LIN {X 0,Y 357.465,Z 383.249,A -85,B 0,C 180,E1 -13742.726,E2 -13742.726} C_VEL
LIN {X 0,Y 362.153,Z 407.547,A -85,B 0,C 180,E1 -13743.635,E2 -13743.635} C_VEL
LIN {X 0,Y 359.928,Z 505.63,A -85,B 0,C 180,E1 -13745.602,E2 -13745.602} C_VEL
LIN {X 0,Y 359.113,Z 520.358,A -85,B 0,C 180,E1 -13746.081,E2 -13746.081} C_VEL
LIN {X 0,Y 358.08,Z 533.693,A -85,B 0,C 180,E1 -13746.737,E2 -13746.737} C_VEL
LIN {X 0,Y 356.818,Z 546.527,A -85,B 0,C 180,E1 -13747.584,E2 -13747.584} C_VEL
LIN {X 0,Y 355.315,Z 560.099,A -85,B 0,C 180,E1 -13748.756,E2 -13748.756} C_VEL
LIN {X 0,Y 353.736,Z 572.534,A -85,B 0,C 180,E1 -13750.111,E2 -13750.111} C_VEL
LIN {X 0,Y 352.276,Z 582.212,A -85,B 0,C 180,E1 -13751.387,E2 -13751.387} C_VEL
LIN {X 0,Y 350.676,Z 592.94,A -85,B 0,C 180,E1 -13753.108,E2 -13753.108} C_VEL
LIN {X 0,Y 349.287,Z 602.41,A -85,B 0,C 180,E1 -13754.974,E2 -13754.974} C_VEL
LIN {X 0,Y 348.307,Z 610.286,A -85,B 0,C 180,E1 -13756.882,E2 -13756.882} C_VEL
LIN {X 0,Y 347.296,Z 617.122,A -85,B 0,C 180,E1 -13758.918,E2 -13758.918} C_VEL
LIN {X 0,Y 346.767,Z 621.834,A -85,B 0,C 180,E1 -13760.671,E2 -13760.671} C_VEL
LIN {X 0,Y 346.34,Z 626.723,A -85,B 0,C 180,E1 -13763.009,E2 -13763.009} C_VEL
LIN {X 0,Y 346.157,Z 630.119,A -85,B 0,C 180,E1 -13765.344,E2 -13765.344} C_VEL
LIN {X 0,Y 346.044,Z 632.123,A -85,B 0,C 180,E1 -13767.674,E2 -13767.674} C_VEL
LIN {X 0,Y 346.074,Z 632.783,A -85,B 0,C 180,E1 -13770.002,E2 -13770.002} C_VEL
LIN {X 0,Y 346.045,Z 632.11,A -85,B 0,C 180,E1 -13772.33,E2 -13772.33} C_VEL
LIN {X 0,Y 346.159,Z 630.094,A -85,B 0,C 180,E1 -13774.66,E2 -13774.66} C_VEL
LIN {X 0,Y 346.372,Z 626.69,A -85,B 0,C 180,E1 -13776.994,E2 -13776.994} C_VEL
LIN {X 0,Y 346.77,Z 621.795,A -85,B 0,C 180,E1 -13779.333,E2 -13779.333} C_VEL
LIN {X 0,Y 347.504,Z 615.257,A -85,B 0,C 180,E1 -13781.67,E2 -13781.67} C_VEL
LIN {X 0,Y 348.587,Z 607.983,A -85,B 0,C 180,E1 -13783.705,E2 -13783.705} C_VEL
LIN {X 0,Y 349.575,Z 600.359,A -85,B 0,C 180,E1 -13785.451,E2 -13785.451} C_VEL
LIN {X 0,Y 350.943,Z 591.212,A -85,B 0,C 180,E1 -13787.182,E2 -13787.182} C_VEL
LIN {X 0,Y 352.599,Z 580.119,A -85,B 0,C 180,E1 -13788.9,E2 -13788.9} C_VEL
LIN {X 0,Y 354.174,Z 568.789,A -85,B 0,C 180,E1 -13790.321,E2 -13790.321} C_VEL
LIN {X 0,Y 355.683,Z 557.277,A -85,B 0,C 180,E1 -13791.497,E2 -13791.497} C_VEL
LIN {X 0,Y 357.075,Z 543.844,A -85,B 0,C 180,E1 -13792.594,E2 -13792.594} C_VEL
LIN {X 0,Y 358.271,Z 530.811,A -85,B 0,C 180,E1 -13793.407,E2 -13793.407} C_VEL
LIN {X 0,Y 359.345,Z 516.257,A -85,B 0,C 180,E1 -13794.059,E2 -13794.059} C_VEL
LIN {X 0,Y 360.003,Z 501.856,A -85,B 0,C 180,E1 -13794.473,E2 -13794.473} C_VEL
LIN {X 0,Y 362.154,Z 407.859,A -85,B 0,C 180,E1 -13796.342,E2 -13796.342} C_VEL
LIN {X 0,Y 358.804,Z 389.741,A -85,B 0,C 180,E1 -13797.02,E2 -13797.02} C_VEL
LIN {X 0,Y 358.775,Z 382.831,A -85,B 0,C 180,E1 -13797.702,E2 -13797.702} C_VEL
LIN {X 0,Y 355.442,Z 371.34,A -85,B 0,C 180,E1 -13799.626,E2 -13799.626} C_VEL
LIN {X 0,Y 352.527,Z 362.364,A -85,B 0,C 180,E1 -13801.555,E2 -13801.555} C_VEL
LIN {X 0,Y 351.134,Z 357.356,A -85,B 0,C 180,E1 -13802.793,E2 -13802.793} C_VEL
LIN {X 0,Y 350.669,Z 355.832,A -85,B 0,C 180,E1 -13803.224,E2 -13803.224} C_VEL
LIN {X 0,Y 348.242,Z 352.609,A -85,B 0,C 180,E1 -13804.76,E2 -13804.76} C_VEL
LIN {X 0,Y 347.783,Z 350.788,A -85,B 0,C 180,E1 -13805.432,E2 -13805.432} C_VEL
LIN {X 0,Y 347.757,Z 350.788,A -85,B 0,C 180,E1 -13808.794,E2 -13808.794} C_VEL
LIN {X 0,Y 347.756,Z 350.79,A -85,B 0,C 180,E1 -13811.831,E2 -13811.831} C_VEL
LIN {X 0,Y 347.711,Z 350.798,A -85,B 0,C 180,E1 -13815.028,E2 -13815.028} C_VEL
LIN {X 0,Y 347.756,Z 350.789,A -85,B 0,C 180,E1 -13818.398,E2 -13818.398} C_VEL
LIN {X 0,Y 347.783,Z 350.968,A -85,B 0,C 180,E1 -13821.833,E2 -13821.833} C_VEL
LIN {X 0,Y 349.99,Z 356.011,A -85,B 0,C 180,E1 -13824.385,E2 -13824.385} C_VEL
LIN {X 0,Y 352.489,Z 361.906,A -85,B 0,C 180,E1 -13826.869,E2 -13826.869} C_VEL
LIN {X 0,Y 355.394,Z 370.388,A -85,B 0,C 180,E1 -13829.806,E2 -13829.806} C_VEL
LIN {X 0,Y 357.469,Z 378.499,A -85,B 0,C 180,E1 -13832.219,E2 -13832.219} C_VEL
LIN {X 0,Y 358.749,Z 385.06,A -85,B 0,C 180,E1 -13833.939,E2 -13833.939} C_VEL
LIN {X 0,Y 360.517,Z 390.055,A -85,B 0,C 180,E1 -13834.446,E2 -13834.446} C_VEL
LIN {X 0,Y 363.882,Z 403.752,A -85,B 0,C 180,E1 -13835.525,E2 -13835.525} C_VEL
LIN {X 0,Y 364.859,Z 409.674,A -85,B 0,C 180,E1 -13835.903,E2 -13835.903} C_VEL
LIN {X 0,Y 359.356,Z 495.934,A -85,B 0,C 180,E1 -13838.676,E2 -13838.676} C_VEL
LIN {X 0,Y 358.366,Z 509.009,A -85,B 0,C 180,E1 -13839.329,E2 -13839.329} C_VEL
LIN {X 0,Y 357.221,Z 521.386,A -85,B 0,C 180,E1 -13840.161,E2 -13840.161} C_VEL
LIN {X 0,Y 355.815,Z 533.988,A -85,B 0,C 180,E1 -13841.279,E2 -13841.279} C_VEL
LIN {X 0,Y 354.377,Z 544.644,A -85,B 0,C 180,E1 -13842.453,E2 -13842.453} C_VEL
LIN {X 0,Y 352.96,Z 554.521,A -85,B 0,C 180,E1 -13843.814,E2 -13843.814} C_VEL
LIN {X 0,Y 351.593,Z 563.035,A -85,B 0,C 180,E1 -13845.235,E2 -13845.235} C_VEL
LIN {X 0,Y 350.232,Z 571.357,A -85,B 0,C 180,E1 -13846.953,E2 -13846.953} C_VEL
LIN {X 0,Y 349.336,Z 577.026,A -85,B 0,C 180,E1 -13848.394,E2 -13848.394} C_VEL
LIN {X 0,Y 348.363,Z 582.532,A -85,B 0,C 180,E1 -13850.126,E2 -13850.126} C_VEL
LIN {X 0,Y 347.582,Z 587.534,A -85,B 0,C 180,E1 -13852.215,E2 -13852.215} C_VEL
LIN {X 0,Y 346.856,Z 590.83,A -85,B 0,C 180,E1 -13854.185,E2 -13854.185} C_VEL
LIN {X 0,Y 346.733,Z 592.108,A -85,B 0,C 180,E1 -13855.35,E2 -13855.35} C_VEL
LIN {X 0,Y 346.66,Z 592.979,A -85,B 0,C 180,E1 -13856.513,E2 -13856.513} C_VEL
LIN {X 0,Y 346.502,Z 593.434,A -85,B 0,C 180,E1 -13857.675,E2 -13857.675} C_VEL
LIN {X 0,Y 346.372,Z 593.414,A -85,B 0,C 180,E1 -13858.837,E2 -13858.837} C_VEL
LIN {X 0,Y 346.288,Z 592.975,A -85,B 0,C 180,E1 -13860,E2 -13860} C_VEL
LIN {X 0,Y 346.263,Z 592.118,A -85,B 0,C 180,E1 -13861.163,E2 -13861.163} C_VEL
LIN {X 0,Y 346.269,Z 590.774,A -85,B 0,C 180,E1 -13862.327,E2 -13862.327} C_VEL
LIN {X 0,Y 346.381,Z 587.926,A -85,B 0,C 180,E1 -13864.072,E2 -13864.072} C_VEL
LIN {X 0,Y 346.518,Z 583.457,A -85,B 0,C 180,E1 -13866.021,E2 -13866.021} C_VEL
LIN {X 0,Y 346.823,Z 577.854,A -85,B 0,C 180,E1 -13867.862,E2 -13867.862} C_VEL
LIN {X 0,Y 347.272,Z 571.051,A -85,B 0,C 180,E1 -13869.611,E2 -13869.611} C_VEL
LIN {X 0,Y 347.827,Z 562.589,A -85,B 0,C 180,E1 -13871.362,E2 -13871.362} C_VEL
LIN {X 0,Y 348.477,Z 553.904,A -85,B 0,C 180,E1 -13872.818,E2 -13872.818} C_VEL
LIN {X 0,Y 349.269,Z 543.265,A -85,B 0,C 180,E1 -13874.27,E2 -13874.27} C_VEL
LIN {X 0,Y 350,Z 531.661,A -85,B 0,C 180,E1 -13875.545,E2 -13875.545} C_VEL
LIN {X 0,Y 350.635,Z 519.537,A -85,B 0,C 180,E1 -13876.596,E2 -13876.596} C_VEL
LIN {X 0,Y 351.426,Z 506.477,A -85,B 0,C 180,E1 -13877.456,E2 -13877.456} C_VEL
LIN {X 0,Y 351.884,Z 492.768,A -85,B 0,C 180,E1 -13878.109,E2 -13878.109} C_VEL
LIN {X 0,Y 352.421,Z 471.978,A -85,B 0,C 180,E1 -13878.72,E2 -13878.72} C_VEL
LIN {X 0,Y 354.249,Z 403.289,A -85,B 0,C 180,E1 -13880.582,E2 -13880.582} C_VEL
LIN {X 0,Y 350.792,Z 379.622,A -85,B 0,C 180,E1 -13881.408,E2 -13881.408} C_VEL
LIN {X 0,Y 351.266,Z 368.636,A -85,B 0,C 180,E1 -13883.588,E2 -13883.588} C_VEL
LIN {X 0,Y 348.86,Z 355.776,A -85,B 0,C 180,E1 -13886.309,E2 -13886.309} C_VEL
LIN {X 0,Y 347.872,Z 350.779,A -85,B 0,C 180,E1 -13887.413,E2 -13887.413} C_VEL
LIN {X 0,Y 347.77,Z 350.789,A -85,B 0,C 180,E1 -13890.346,E2 -13890.346} C_VEL
LIN {X 0,Y 347.751,Z 350.794,A -85,B 0,C 180,E1 -13894.463,E2 -13894.463} C_VEL
LIN {X 0,Y 347.769,Z 350.792,A -85,B 0,C 180,E1 -13897.986,E2 -13897.986} C_VEL
LIN {X 0,Y 347.75,Z 350.796,A -85,B 0,C 180,E1 -13901.831,E2 -13901.831} C_VEL
LIN {X 0,Y 347.711,Z 350.798,A -85,B 0,C 180,E1 -13905.026,E2 -13905.026} C_VEL
LIN {X 0,Y 347.747,Z 350.792,A -85,B 0,C 180,E1 -13908.398,E2 -13908.398} C_VEL
LIN {X 0,Y 347.76,Z 350.792,A -85,B 0,C 180,E1 -13912.677,E2 -13912.677} C_VEL
LIN {X 0,Y 347.753,Z 350.792,A -85,B 0,C 180,E1 -13915.955,E2 -13915.955} C_VEL
LIN {X 0,Y 347.774,Z 350.865,A -85,B 0,C 180,E1 -13918.138,E2 -13918.138} C_VEL
LIN {X 0,Y 350.38,Z 361.692,A -85,B 0,C 180,E1 -13921.222,E2 -13921.222} C_VEL
LIN {X 0,Y 350.969,Z 364.366,A -85,B 0,C 180,E1 -13921.948,E2 -13921.948} C_VEL
LIN {X 0,Y 359.378,Z 384.591,A -85,B 0,C 180,E1 -13923.108,E2 -13923.108} C_VEL
LIN {X 0,Y 362.312,Z 400.294,A -85,B 0,C 180,E1 -13923.685,E2 -13923.685} C_VEL
LIN {X 0,Y 360.052,Z 498.393,A -85,B 0,C 180,E1 -13925.646,E2 -13925.646} C_VEL
LIN {X 0,Y 359.513,Z 509.877,A -85,B 0,C 180,E1 -13925.991,E2 -13925.991} C_VEL
LIN {X 0,Y 358.474,Z 523.814,A -85,B 0,C 180,E1 -13926.607,E2 -13926.607} C_VEL
LIN {X 0,Y 357.377,Z 537.009,A -85,B 0,C 180,E1 -13927.426,E2 -13927.426} C_VEL
LIN {X 0,Y 356.097,Z 549.518,A -85,B 0,C 180,E1 -13928.432,E2 -13928.432} C_VEL
LIN {X 0,Y 354.541,Z 562.109,A -85,B 0,C 180,E1 -13929.701,E2 -13929.701} C_VEL
LIN {X 0,Y 352.879,Z 573.479,A -85,B 0,C 180,E1 -13931.115,E2 -13931.115} C_VEL
LIN {X 0,Y 351.531,Z 582.899,A -85,B 0,C 180,E1 -13932.548,E2 -13932.548} C_VEL
LIN {X 0,Y 350.087,Z 592.37,A -85,B 0,C 180,E1 -13934.274,E2 -13934.274} C_VEL
LIN {X 0,Y 348.912,Z 601.393,A -85,B 0,C 180,E1 -13936.308,E2 -13936.308} C_VEL
LIN {X 0,Y 347.753,Z 608.668,A -85,B 0,C 180,E1 -13938.339,E2 -13938.339} C_VEL
LIN {X 0,Y 347.139,Z 613.758,A -85,B 0,C 180,E1 -13940.089,E2 -13940.089} C_VEL
LIN {X 0,Y 346.562,Z 619.033,A -85,B 0,C 180,E1 -13942.424,E2 -13942.424} C_VEL
LIN {X 0,Y 346.346,Z 621.974,A -85,B 0,C 180,E1 -13944.175,E2 -13944.175} C_VEL
LIN {X 0,Y 346.16,Z 624.682,A -85,B 0,C 180,E1 -13946.506,E2 -13946.506} C_VEL
LIN {X 0,Y 346.06,Z 626.041,A -85,B 0,C 180,E1 -13948.835,E2 -13948.835} C_VEL
LIN {X 0,Y 346.06,Z 626.076,A -85,B 0,C 180,E1 -13951.162,E2 -13951.162} C_VEL
LIN {X 0,Y 346.158,Z 624.787,A -85,B 0,C 180,E1 -13953.49,E2 -13953.49} C_VEL
LIN {X 0,Y 346.337,Z 622.141,A -85,B 0,C 180,E1 -13955.822,E2 -13955.822} C_VEL
LIN {X 0,Y 346.663,Z 618.067,A -85,B 0,C 180,E1 -13958.157,E2 -13958.157} C_VEL
LIN {X 0,Y 347.305,Z 612.441,A -85,B 0,C 180,E1 -13960.492,E2 -13960.492} C_VEL
LIN {X 0,Y 348.174,Z 606.094,A -85,B 0,C 180,E1 -13962.531,E2 -13962.531} C_VEL
LIN {X 0,Y 348.426,Z 604.675,A -85,B 0,C 180,E1 -13962.933,E2 -13962.933} C_VEL
LIN {X 0,Y 348.241,Z 601.627,A -85,B 0,C 180,E1 -13963.764,E2 -13963.764} C_VEL
LIN {X 0,Y 346.181,Z 596.49,A -85,B 0,C 180,E1 -13965.123,E2 -13965.123} C_VEL
LIN {X 0,Y 344.187,Z 590.868,A -85,B 0,C 180,E1 -13966.44,E2 -13966.44} C_VEL
LIN {X 0,Y 344.099,Z 587.06,A -85,B 0,C 180,E1 -13967.192,E2 -13967.192} C_VEL
LIN {X 0,Y 345.798,Z 576.239,A -85,B 0,C 180,E1 -13968.975,E2 -13968.975} C_VEL
LIN {X 0,Y 347.416,Z 565.469,A -85,B 0,C 180,E1 -13970.421,E2 -13970.421} C_VEL
LIN {X 0,Y 349.017,Z 554.043,A -85,B 0,C 180,E1 -13971.675,E2 -13971.675} C_VEL
LIN {X 0,Y 350.388,Z 541.472,A -85,B 0,C 180,E1 -13972.796,E2 -13972.796} C_VEL
LIN {X 0,Y 351.677,Z 528.19,A -85,B 0,C 180,E1 -13973.713,E2 -13973.713} C_VEL
LIN {X 0,Y 352.764,Z 514.34,A -85,B 0,C 180,E1 -13974.416,E2 -13974.416} C_VEL
LIN {X 0,Y 353.581,Z 499.725,A -85,B 0,C 180,E1 -13974.904,E2 -13974.904} C_VEL
LIN {X 0,Y 355.998,Z 400.884,A -85,B 0,C 180,E1 -13976.915,E2 -13976.915} C_VEL
LIN {X 0,Y 353.055,Z 386.375,A -85,B 0,C 180,E1 -13977.484,E2 -13977.484} C_VEL
LIN {X 0,Y 345.906,Z 369.454,A -85,B 0,C 180,E1 -13978.494,E2 -13978.494} C_VEL
LIN {X 0,Y 343.732,Z 364.278,A -85,B 0,C 180,E1 -13978.843,E2 -13978.843} C_VEL
LIN {X 0,Y 341.03,Z 353.043,A -85,B 0,C 180,E1 -13982.107,E2 -13982.107} C_VEL
LIN {X 0,Y 340.697,Z 351.677,A -85,B 0,C 180,E1 -13982.52,E2 -13982.52} C_VEL
LIN {X 0,Y 340.711,Z 351.675,A -85,B 0,C 180,E1 -13985.277,E2 -13985.277} C_VEL
LIN {X 0,Y 340.686,Z 351.674,A -85,B 0,C 180,E1 -13988.381,E2 -13988.381} C_VEL
LIN {X 0,Y 340.681,Z 351.672,A -85,B 0,C 180,E1 -13992.042,E2 -13992.042} C_VEL
LIN {X 0,Y 340.641,Z 351.677,A -85,B 0,C 180,E1 -13996.226,E2 -13996.226} C_VEL
LIN {X 0,Y 340.661,Z 351.675,A -85,B 0,C 180,E1 -13998.686,E2 -13998.686} C_VEL
LIN {X 0,Y 340.708,Z 351.657,A -85,B 0,C 180,E1 -14001.769,E2 -14001.769} C_VEL
LIN {X 0,Y 340.712,Z 351.665,A -85,B 0,C 180,E1 -14005.594,E2 -14005.594} C_VEL
LIN {X 0,Y 340.678,Z 351.668,A -85,B 0,C 180,E1 -14008.953,E2 -14008.953} C_VEL
LIN {X 0,Y 340.698,Z 351.651,A -85,B 0,C 180,E1 -14013.011,E2 -14013.011} C_VEL
LIN {X 0,Y 340.731,Z 351.662,A -85,B 0,C 180,E1 -14015.636,E2 -14015.636} C_VEL
LIN {X 0,Y 340.715,Z 351.655,A -85,B 0,C 180,E1 -14019.472,E2 -14019.472} C_VEL
LIN {X 0,Y 340.779,Z 351.644,A -85,B 0,C 180,E1 -14021.98,E2 -14021.98} C_VEL
LIN {X 0,Y 340.839,Z 351.65,A -85,B 0,C 180,E1 -14025.716,E2 -14025.716} C_VEL
LIN {X 0,Y 340.833,Z 351.652,A -85,B 0,C 180,E1 -14029.305,E2 -14029.305} C_VEL
LIN {X 0,Y 340.983,Z 351.637,A -85,B 0,C 180,E1 -14032.896,E2 -14032.896} C_VEL
LIN {X 0,Y 340.802,Z 351.65,A -85,B 0,C 180,E1 -14035.268,E2 -14035.268} C_VEL
LIN {X 0,Y 341.114,Z 351.617,A -85,B 0,C 180,E1 -14037.638,E2 -14037.638} C_VEL
LIN {X 0,Y 341.097,Z 351.62,A -85,B 0,C 180,E1 -14041.181,E2 -14041.181} C_VEL
LIN {X 0,Y 341.111,Z 351.622,A -85,B 0,C 180,E1 -14042.362,E2 -14042.362} C_VEL
LIN {X 0,Y 341,Z 351.631,A -85,B 0,C 180,E1 -14045.915,E2 -14045.915} C_VEL
LIN {X 0,Y 340.949,Z 351.635,A -85,B 0,C 180,E1 -14048.356,E2 -14048.356} C_VEL
LIN {X 0,Y 340.83,Z 351.653,A -85,B 0,C 180,E1 -14051.9,E2 -14051.9} C_VEL
LIN {X 0,Y 340.803,Z 351.655,A -85,B 0,C 180,E1 -14055.55,E2 -14055.55} C_VEL
LIN {X 0,Y 340.72,Z 351.665,A -85,B 0,C 180,E1 -14059.271,E2 -14059.271} C_VEL
LIN {X 0,Y 340.687,Z 351.655,A -85,B 0,C 180,E1 -14063.076,E2 -14063.076} C_VEL
LIN {X 0,Y 340.697,Z 351.666,A -85,B 0,C 180,E1 -14066.989,E2 -14066.989} C_VEL
LIN {X 0,Y 340.678,Z 351.672,A -85,B 0,C 180,E1 -14071.047,E2 -14071.047} C_VEL
LIN {X 0,Y 340.703,Z 351.669,A -85,B 0,C 180,E1 -14075.281,E2 -14075.281} C_VEL
LIN {X 0,Y 340.681,Z 351.672,A -85,B 0,C 180,E1 -14078.384,E2 -14078.384} C_VEL
LIN {X 0,Y 340.679,Z 351.674,A -85,B 0,C 180,E1 -14082.045,E2 -14082.045} C_VEL
LIN {X 0,Y 340.639,Z 351.68,A -85,B 0,C 180,E1 -14086.229,E2 -14086.229} C_VEL
LIN {X 0,Y 340.658,Z 351.68,A -85,B 0,C 180,E1 -14088.689,E2 -14088.689} C_VEL
LIN {X 0,Y 340.709,Z 351.674,A -85,B 0,C 180,E1 -14091.772,E2 -14091.772} C_VEL
LIN {X 0,Y 340.714,Z 351.671,A -85,B 0,C 180,E1 -14095.598,E2 -14095.598} C_VEL
LIN {X 0,Y 340.718,Z 351.759,A -85,B 0,C 180,E1 -14096.257,E2 -14096.257} C_VEL
LIN {X 0,Y 343.521,Z 363.282,A -85,B 0,C 180,E1 -14099.536,E2 -14099.536} C_VEL
LIN {X 0,Y 345.053,Z 370.085,A -85,B 0,C 180,E1 -14101.355,E2 -14101.355} C_VEL
LIN {X 0,Y 351.366,Z 385.442,A -85,B 0,C 180,E1 -14102.263,E2 -14102.263} C_VEL
LIN {X 0,Y 355.832,Z 409.247,A -85,B 0,C 180,E1 -14103.168,E2 -14103.168} C_VEL
LIN {X 0,Y 353.438,Z 507.052,A -85,B 0,C 180,E1 -14105.164,E2 -14105.164} C_VEL
LIN {X 0,Y 352.525,Z 521.861,A -85,B 0,C 180,E1 -14105.684,E2 -14105.684} C_VEL
LIN {X 0,Y 351.323,Z 535.9,A -85,B 0,C 180,E1 -14106.419,E2 -14106.419} C_VEL
LIN {X 0,Y 349.916,Z 549.82,A -85,B 0,C 180,E1 -14107.413,E2 -14107.413} C_VEL
LIN {X 0,Y 348.4,Z 562.583,A -85,B 0,C 180,E1 -14108.59,E2 -14108.59} C_VEL
LIN {X 0,Y 346.649,Z 574.815,A -85,B 0,C 180,E1 -14109.996,E2 -14109.996} C_VEL
LIN {X 0,Y 344.939,Z 585.993,A -85,B 0,C 180,E1 -14111.593,E2 -14111.593} C_VEL
LIN {X 0,Y 343.34,Z 596.02,A -85,B 0,C 180,E1 -14113.349,E2 -14113.349} C_VEL
LIN {X 0,Y 341.994,Z 605.417,A -85,B 0,C 180,E1 -14115.381,E2 -14115.381} C_VEL
LIN {X 0,Y 340.882,Z 613.322,A -85,B 0,C 180,E1 -14117.5,E2 -14117.5} C_VEL
LIN {X 0,Y 340.094,Z 618.721,A -85,B 0,C 180,E1 -14119.283,E2 -14119.283} C_VEL
LIN {X 0,Y 339.495,Z 624.407,A -85,B 0,C 180,E1 -14121.67,E2 -14121.67} C_VEL
LIN {X 0,Y 339.168,Z 628.534,A -85,B 0,C 180,E1 -14124.055,E2 -14124.055} C_VEL
LIN {X 0,Y 339.043,Z 631.224,A -85,B 0,C 180,E1 -14126.436,E2 -14126.436} C_VEL
LIN {X 0,Y 338.954,Z 632.552,A -85,B 0,C 180,E1 -14128.814,E2 -14128.814} C_VEL
LIN {X 0,Y 338.954,Z 632.546,A -85,B 0,C 180,E1 -14131.19,E2 -14131.19} C_VEL
LIN {X 0,Y 339.044,Z 631.204,A -85,B 0,C 180,E1 -14133.567,E2 -14133.567} C_VEL
LIN {X 0,Y 339.17,Z 628.503,A -85,B 0,C 180,E1 -14135.949,E2 -14135.949} C_VEL
LIN {X 0,Y 339.498,Z 624.369,A -85,B 0,C 180,E1 -14138.334,E2 -14138.334} C_VEL
LIN {X 0,Y 340.097,Z 618.674,A -85,B 0,C 180,E1 -14140.72,E2 -14140.72} C_VEL
LIN {X 0,Y 341.017,Z 612.251,A -85,B 0,C 180,E1 -14142.802,E2 -14142.802} C_VEL
LIN {X 0,Y 342.168,Z 604.024,A -85,B 0,C 180,E1 -14144.94,E2 -14144.94} C_VEL
LIN {X 0,Y 343.353,Z 595.927,A -85,B 0,C 180,E1 -14146.654,E2 -14146.654} C_VEL
LIN {X 0,Y 344.968,Z 585.88,A -85,B 0,C 180,E1 -14148.41,E2 -14148.41} C_VEL
LIN {X 0,Y 346.631,Z 574.668,A -85,B 0,C 180,E1 -14150.009,E2 -14150.009} C_VEL
LIN {X 0,Y 348.365,Z 562.362,A -85,B 0,C 180,E1 -14151.419,E2 -14151.419} C_VEL
LIN {X 0,Y 349.939,Z 549.589,A -85,B 0,C 180,E1 -14152.589,E2 -14152.589} C_VEL
LIN {X 0,Y 351.207,Z 536.743,A -85,B 0,C 180,E1 -14153.515,E2 -14153.515} C_VEL
LIN {X 0,Y 352.451,Z 522.994,A -85,B 0,C 180,E1 -14154.247,E2 -14154.247} C_VEL
LIN {X 0,Y 353.287,Z 508.773,A -85,B 0,C 180,E1 -14154.773,E2 -14154.773} C_VEL
LIN {X 0,Y 354.304,Z 475.141,A -85,B 0,C 180,E1 -14155.482,E2 -14155.482} C_VEL
LIN {X 0,Y 355.688,Z 408.276,A -85,B 0,C 180,E1 -14156.847,E2 -14156.847} C_VEL
LIN {X 0,Y 353.441,Z 395.591,A -85,B 0,C 180,E1 -14157.341,E2 -14157.341} C_VEL
LIN {X 0,Y 353.614,Z 387.326,A -85,B 0,C 180,E1 -14158.142,E2 -14158.142} C_VEL
LIN {X 0,Y 353.492,Z 385.813,A -85,B 0,C 180,E1 -14158.327,E2 -14158.327} C_VEL
LIN {X 0,Y 350.231,Z 374.456,A -85,B 0,C 180,E1 -14160.36,E2 -14160.36} C_VEL
LIN {X 0,Y 347.43,Z 364.788,A -85,B 0,C 180,E1 -14162.549,E2 -14162.549} C_VEL
LIN {X 0,Y 346.783,Z 362.458,A -85,B 0,C 180,E1 -14163.176,E2 -14163.176} C_VEL
LIN {X 0,Y 346.13,Z 361.067,A -85,B 0,C 180,E1 -14163.645,E2 -14163.645} C_VEL
LIN {X 0,Y 344.309,Z 358.527,A -85,B 0,C 180,E1 -14164.859,E2 -14164.859} C_VEL
LIN {X 0,Y 343.174,Z 356.184,A -85,B 0,C 180,E1 -14165.937,E2 -14165.937} C_VEL
LIN {X 0,Y 341.539,Z 354.187,A -85,B 0,C 180,E1 -14167.376,E2 -14167.376} C_VEL
LIN {X 0,Y 340.714,Z 351.667,A -85,B 0,C 180,E1 -14169.108,E2 -14169.108} C_VEL
LIN {X 0,Y 340.681,Z 351.672,A -85,B 0,C 180,E1 -14172.905,E2 -14172.905} C_VEL
LIN {X 0,Y 340.681,Z 351.674,A -85,B 0,C 180,E1 -14177.097,E2 -14177.097} C_VEL
LIN {X 0,Y 340.734,Z 351.761,A -85,B 0,C 180,E1 -14178.33,E2 -14178.33} C_VEL
LIN {X 0,Y 341.693,Z 354.447,A -85,B 0,C 180,E1 -14180.386,E2 -14180.386} C_VEL
LIN {X 0,Y 343.059,Z 356.792,A -85,B 0,C 180,E1 -14182.078,E2 -14182.078} C_VEL
LIN {X 0,Y 345.102,Z 361.499,A -85,B 0,C 180,E1 -14184.55,E2 -14184.55} C_VEL
LIN {X 0,Y 347.264,Z 366.901,A -85,B 0,C 180,E1 -14186.878,E2 -14186.878} C_VEL
LIN {X 0,Y 349.851,Z 374.925,A -85,B 0,C 180,E1 -14189.749,E2 -14189.749} C_VEL
LIN {X 0,Y 351.742,Z 382.879,A -85,B 0,C 180,E1 -14192.175,E2 -14192.175} C_VEL
LIN {X 0,Y 352.347,Z 385.665,A -85,B 0,C 180,E1 -14192.922,E2 -14192.922} C_VEL
LIN {X 0,Y 355.225,Z 392.184,A -85,B 0,C 180,E1 -14193.724,E2 -14193.724} C_VEL
LIN {X 0,Y 358.347,Z 405.235,A -85,B 0,C 180,E1 -14194.815,E2 -14194.815} C_VEL
LIN {X 0,Y 359.33,Z 410.888,A -85,B 0,C 180,E1 -14195.211,E2 -14195.211} C_VEL
LIN {X 0,Y 353.408,Z 496.747,A -85,B 0,C 180,E1 -14198.069,E2 -14198.069} C_VEL
LIN {X 0,Y 352.236,Z 510.74,A -85,B 0,C 180,E1 -14198.799,E2 -14198.799} C_VEL
LIN {X 0,Y 351.024,Z 522.696,A -85,B 0,C 180,E1 -14199.643,E2 -14199.643} C_VEL
LIN {X 0,Y 349.501,Z 535.21,A -85,B 0,C 180,E1 -14200.791,E2 -14200.791} C_VEL
LIN {X 0,Y 348.087,Z 544.698,A -85,B 0,C 180,E1 -14201.858,E2 -14201.858} C_VEL
LIN {X 0,Y 346.636,Z 554.379,A -85,B 0,C 180,E1 -14203.207,E2 -14203.207} C_VEL
LIN {X 0,Y 344.879,Z 564.519,A -85,B 0,C 180,E1 -14204.941,E2 -14204.941} C_VEL
LIN {X 0,Y 343.437,Z 572.571,A -85,B 0,C 180,E1 -14206.69,E2 -14206.69} C_VEL
LIN {X 0,Y 342.484,Z 578.088,A -85,B 0,C 180,E1 -14208.158,E2 -14208.158} C_VEL
LIN {X 0,Y 341.438,Z 583.452,A -85,B 0,C 180,E1 -14209.924,E2 -14209.924} C_VEL
LIN {X 0,Y 340.698,Z 587.6,A -85,B 0,C 180,E1 -14211.698,E2 -14211.698} C_VEL
LIN {X 0,Y 340.282,Z 589.771,A -85,B 0,C 180,E1 -14212.882,E2 -14212.882} C_VEL
LIN {X 0,Y 339.829,Z 591.443,A -85,B 0,C 180,E1 -14214.065,E2 -14214.065} C_VEL
LIN {X 0,Y 339.668,Z 592.667,A -85,B 0,C 180,E1 -14215.253,E2 -14215.253} C_VEL
LIN {X 0,Y 339.582,Z 593.477,A -85,B 0,C 180,E1 -14216.44,E2 -14216.44} C_VEL
LIN {X 0,Y 339.417,Z 593.824,A -85,B 0,C 180,E1 -14217.627,E2 -14217.627} C_VEL
LIN {X 0,Y 339.281,Z 593.742,A -85,B 0,C 180,E1 -14218.813,E2 -14218.813} C_VEL
LIN {X 0,Y 339.194,Z 593.245,A -85,B 0,C 180,E1 -14220,E2 -14220} C_VEL
LIN {X 0,Y 339.165,Z 592.283,A -85,B 0,C 180,E1 -14221.187,E2 -14221.187} C_VEL
LIN {X 0,Y 339.176,Z 590.872,A -85,B 0,C 180,E1 -14222.375,E2 -14222.375} C_VEL
LIN {X 0,Y 339.313,Z 587.905,A -85,B 0,C 180,E1 -14224.157,E2 -14224.157} C_VEL
LIN {X 0,Y 339.43,Z 583.828,A -85,B 0,C 180,E1 -14225.942,E2 -14225.942} C_VEL
LIN {X 0,Y 339.714,Z 578.533,A -85,B 0,C 180,E1 -14227.728,E2 -14227.728} C_VEL
LIN {X 0,Y 340.139,Z 571.809,A -85,B 0,C 180,E1 -14229.515,E2 -14229.515} C_VEL
LIN {X 0,Y 340.715,Z 563.416,A -85,B 0,C 180,E1 -14231.301,E2 -14231.301} C_VEL
LIN {X 0,Y 341.37,Z 554.859,A -85,B 0,C 180,E1 -14232.787,E2 -14232.787} C_VEL
LIN {X 0,Y 342.138,Z 544.343,A -85,B 0,C 180,E1 -14234.27,E2 -14234.27} C_VEL
LIN {X 0,Y 342.901,Z 532.783,A -85,B 0,C 180,E1 -14235.59,E2 -14235.59} C_VEL
LIN {X 0,Y 343.557,Z 521.096,A -85,B 0,C 180,E1 -14236.642,E2 -14236.642} C_VEL
LIN {X 0,Y 344.295,Z 508.539,A -85,B 0,C 180,E1 -14237.523,E2 -14237.523} C_VEL
LIN {X 0,Y 344.846,Z 494.714,A -85,B 0,C 180,E1 -14238.223,E2 -14238.223} C_VEL
LIN {X 0,Y 345.324,Z 478.996,A -85,B 0,C 180,E1 -14238.734,E2 -14238.734} C_VEL
LIN {X 0,Y 347.315,Z 403.908,A -85,B 0,C 180,E1 -14240.832,E2 -14240.832} C_VEL
LIN {X 0,Y 343.829,Z 379.814,A -85,B 0,C 180,E1 -14241.706,E2 -14241.706} C_VEL
LIN {X 0,Y 344.308,Z 370.365,A -85,B 0,C 180,E1 -14243.594,E2 -14243.594} C_VEL
LIN {X 0,Y 342.729,Z 361.219,A -85,B 0,C 180,E1 -14245.54,E2 -14245.54} C_VEL
LIN {X 0,Y 340.854,Z 351.653,A -85,B 0,C 180,E1 -14247.643,E2 -14247.643} C_VEL
LIN {X 0,Y 340.71,Z 351.665,A -85,B 0,C 180,E1 -14251.044,E2 -14251.044} C_VEL
LIN {X 0,Y 340.724,Z 351.668,A -85,B 0,C 180,E1 -14255.278,E2 -14255.278} C_VEL
LIN {X 0,Y 340.699,Z 351.67,A -85,B 0,C 180,E1 -14258.382,E2 -14258.382} C_VEL
LIN {X 0,Y 340.7,Z 351.673,A -85,B 0,C 180,E1 -14262.044,E2 -14262.044} C_VEL
LIN {X 0,Y 340.657,Z 351.677,A -85,B 0,C 180,E1 -14266.226,E2 -14266.226} C_VEL
LIN {X 0,Y 340.676,Z 351.673,A -85,B 0,C 180,E1 -14268.687,E2 -14268.687} C_VEL
LIN {X 0,Y 340.724,Z 351.669,A -85,B 0,C 180,E1 -14271.77,E2 -14271.77} C_VEL
LIN {X 0,Y 340.727,Z 351.664,A -85,B 0,C 180,E1 -14275.595,E2 -14275.595} C_VEL
LIN {X 0,Y 340.705,Z 351.822,A -85,B 0,C 180,E1 -14277.639,E2 -14277.639} C_VEL
LIN {X 0,Y 343.154,Z 361.77,A -85,B 0,C 180,E1 -14280.557,E2 -14280.557} C_VEL
LIN {X 0,Y 343.741,Z 364.378,A -85,B 0,C 180,E1 -14281.296,E2 -14281.296} C_VEL
LIN {X 0,Y 352.365,Z 384.774,A -85,B 0,C 180,E1 -14282.53,E2 -14282.53} C_VEL
LIN {X 0,Y 353.759,Z 389.105,A -85,B 0,C 180,E1 -14282.745,E2 -14282.745} C_VEL
LIN {X 0,Y 355.947,Z 401.083,A -85,B 0,C 180,E1 -14283.193,E2 -14283.193} C_VEL
LIN {X 0,Y 353.61,Z 498.481,A -85,B 0,C 180,E1 -14285.173,E2 -14285.173} C_VEL
LIN {X 0,Y 353.042,Z 509.957,A -85,B 0,C 180,E1 -14285.522,E2 -14285.522} C_VEL
LIN {X 0,Y 351.971,Z 523.891,A -85,B 0,C 180,E1 -14286.148,E2 -14286.148} C_VEL
LIN {X 0,Y 350.826,Z 537.083,A -85,B 0,C 180,E1 -14286.981,E2 -14286.981} C_VEL
LIN {X 0,Y 349.487,Z 549.698,A -85,B 0,C 180,E1 -14288.013,E2 -14288.013} C_VEL
LIN {X 0,Y 347.89,Z 562.18,A -85,B 0,C 180,E1 -14289.295,E2 -14289.295} C_VEL
LIN {X 0,Y 346.154,Z 573.55,A -85,B 0,C 180,E1 -14290.734,E2 -14290.734} C_VEL
LIN {X 0,Y 344.755,Z 582.97,A -85,B 0,C 180,E1 -14292.193,E2 -14292.193} C_VEL
LIN {X 0,Y 343.222,Z 592.44,A -85,B 0,C 180,E1 -14293.952,E2 -14293.952} C_VEL
LIN {X 0,Y 341.993,Z 601.463,A -85,B 0,C 180,E1 -14296.025,E2 -14296.025} C_VEL
LIN {X 0,Y 340.761,Z 608.737,A -85,B 0,C 180,E1 -14298.096,E2 -14298.096} C_VEL
LIN {X 0,Y 340.119,Z 613.827,A -85,B 0,C 180,E1 -14299.882,E2 -14299.882} C_VEL
LIN {X 0,Y 339.511,Z 619.101,A -85,B 0,C 180,E1 -14302.266,E2 -14302.266} C_VEL
LIN {X 0,Y 339.28,Z 622.042,A -85,B 0,C 180,E1 -14304.053,E2 -14304.053} C_VEL
LIN {X 0,Y 339.089,Z 624.75,A -85,B 0,C 180,E1 -14306.433,E2 -14306.433} C_VEL
LIN {X 0,Y 338.966,Z 626.108,A -85,B 0,C 180,E1 -14308.81,E2 -14308.81} C_VEL
LIN {X 0,Y 338.966,Z 626.143,A -85,B 0,C 180,E1 -14311.186,E2 -14311.186} C_VEL
LIN {X 0,Y 339.086,Z 624.853,A -85,B 0,C 180,E1 -14313.563,E2 -14313.563} C_VEL
LIN {X 0,Y 339.257,Z 622.208,A -85,B 0,C 180,E1 -14315.943,E2 -14315.943} C_VEL
LIN {X 0,Y 339.608,Z 618.134,A -85,B 0,C 180,E1 -14318.327,E2 -14318.327} C_VEL
LIN {X 0,Y 340.307,Z 612.507,A -85,B 0,C 180,E1 -14320.71,E2 -14320.71} C_VEL
LIN {X 0,Y 341.237,Z 606.159,A -85,B 0,C 180,E1 -14322.789,E2 -14322.789} C_VEL
LIN {X 0,Y 342.229,Z 599.638,A -85,B 0,C 180,E1 -14324.532,E2 -14324.532} C_VEL
LIN {X 0,Y 343.394,Z 591.633,A -85,B 0,C 180,E1 -14326.312,E2 -14326.312} C_VEL
LIN {X 0,Y 344.099,Z 587.06,A -85,B 0,C 180,E1 -14327.192,E2 -14327.192} C_VEL
LIN {X 0,Y 344.07,Z 583.132,A -85,B 0,C 180,E1 -14327.923,E2 -14327.923} C_VEL
LIN {X 0,Y 342.376,Z 576.539,A -85,B 0,C 180,E1 -14329.129,E2 -14329.129} C_VEL
LIN {X 0,Y 340.771,Z 569.597,A -85,B 0,C 180,E1 -14330.281,E2 -14330.281} C_VEL
LIN {X 0,Y 340.855,Z 564.978,A -85,B 0,C 180,E1 -14330.907,E2 -14330.907} C_VEL
LIN {X 0,Y 342.556,Z 553.079,A -85,B 0,C 180,E1 -14332.22,E2 -14332.22} C_VEL
LIN {X 0,Y 343.867,Z 541.426,A -85,B 0,C 180,E1 -14333.263,E2 -14333.263} C_VEL
LIN {X 0,Y 345.205,Z 528.249,A -85,B 0,C 180,E1 -14334.185,E2 -14334.185} C_VEL
LIN {X 0,Y 346.319,Z 514.395,A -85,B 0,C 180,E1 -14334.901,E2 -14334.901} C_VEL
LIN {X 0,Y 347.168,Z 499.771,A -85,B 0,C 180,E1 -14335.397,E2 -14335.397} C_VEL
LIN {X 0,Y 349.677,Z 402.324,A -85,B 0,C 180,E1 -14337.411,E2 -14337.411} C_VEL
LIN {X 0,Y 347.103,Z 389.177,A -85,B 0,C 180,E1 -14337.933,E2 -14337.933} C_VEL
LIN {X 0,Y 339.774,Z 371.607,A -85,B 0,C 180,E1 -14339.007,E2 -14339.007} C_VEL
LIN {X 0,Y 336.54,Z 364.418,A -85,B 0,C 180,E1 -14339.501,E2 -14339.501} C_VEL
LIN {X 0,Y 333.652,Z 352.554,A -85,B 0,C 180,E1 -14343.068,E2 -14343.068} C_VEL
LIN {X 0,Y 333.668,Z 352.548,A -85,B 0,C 180,E1 -14346.137,E2 -14346.137} C_VEL
LIN {X 0,Y 333.594,Z 352.556,A -85,B 0,C 180,E1 -14349.197,E2 -14349.197} C_VEL
LIN {X 0,Y 333.617,Z 352.552,A -85,B 0,C 180,E1 -14352.497,E2 -14352.497} C_VEL
LIN {X 0,Y 333.585,Z 352.555,A -85,B 0,C 180,E1 -14355.953,E2 -14355.953} C_VEL
LIN {X 0,Y 333.592,Z 352.557,A -85,B 0,C 180,E1 -14359.323,E2 -14359.323} C_VEL
LIN {X 0,Y 333.652,Z 352.543,A -85,B 0,C 180,E1 -14363.167,E2 -14363.167} C_VEL
LIN {X 0,Y 333.663,Z 352.544,A -85,B 0,C 180,E1 -14365.34,E2 -14365.34} C_VEL
LIN {X 0,Y 333.615,Z 352.54,A -85,B 0,C 180,E1 -14368.22,E2 -14368.22} C_VEL
LIN {X 0,Y 333.637,Z 352.548,A -85,B 0,C 180,E1 -14371.021,E2 -14371.021} C_VEL
LIN {X 0,Y 333.683,Z 352.535,A -85,B 0,C 180,E1 -14375.087,E2 -14375.087} C_VEL
LIN {X 0,Y 333.649,Z 352.537,A -85,B 0,C 180,E1 -14379.017,E2 -14379.017} C_VEL
LIN {X 0,Y 333.727,Z 352.519,A -85,B 0,C 180,E1 -14381.586,E2 -14381.586} C_VEL
LIN {X 0,Y 333.795,Z 352.528,A -85,B 0,C 180,E1 -14385.576,E2 -14385.576} C_VEL
LIN {X 0,Y 333.802,Z 352.529,A -85,B 0,C 180,E1 -14389.077,E2 -14389.077} C_VEL
LIN {X 0,Y 333.939,Z 352.515,A -85,B 0,C 180,E1 -14392.746,E2 -14392.746} C_VEL
LIN {X 0,Y 333.768,Z 352.526,A -85,B 0,C 180,E1 -14395.168,E2 -14395.168} C_VEL
LIN {X 0,Y 334.055,Z 352.497,A -85,B 0,C 180,E1 -14397.588,E2 -14397.588} C_VEL
LIN {X 0,Y 334.065,Z 352.496,A -85,B 0,C 180,E1 -14401.205,E2 -14401.205} C_VEL
LIN {X 0,Y 333.791,Z 352.526,A -85,B 0,C 180,E1 -14403.621,E2 -14403.621} C_VEL
LIN {X 0,Y 333.974,Z 352.507,A -85,B 0,C 180,E1 -14406.04,E2 -14406.04} C_VEL
LIN {X 0,Y 333.898,Z 352.513,A -85,B 0,C 180,E1 -14408.473,E2 -14408.473} C_VEL
LIN {X 0,Y 333.772,Z 352.531,A -85,B 0,C 180,E1 -14412.155,E2 -14412.155} C_VEL
LIN {X 0,Y 333.759,Z 352.534,A -85,B 0,C 180,E1 -14415.887,E2 -14415.887} C_VEL
LIN {X 0,Y 333.71,Z 352.543,A -85,B 0,C 180,E1 -14418.618,E2 -14418.618} C_VEL
LIN {X 0,Y 333.635,Z 352.53,A -85,B 0,C 180,E1 -14422.282,E2 -14422.282} C_VEL
LIN {X 0,Y 333.644,Z 352.548,A -85,B 0,C 180,E1 -14425.079,E2 -14425.079} C_VEL
LIN {X 0,Y 333.617,Z 352.535,A -85,B 0,C 180,E1 -14428.981,E2 -14428.981} C_VEL
LIN {X 0,Y 333.63,Z 352.549,A -85,B 0,C 180,E1 -14432.588,E2 -14432.588} C_VEL
LIN {X 0,Y 333.661,Z 352.546,A -85,B 0,C 180,E1 -14436.141,E2 -14436.141} C_VEL
LIN {X 0,Y 333.59,Z 352.555,A -85,B 0,C 180,E1 -14439.2,E2 -14439.2} C_VEL
LIN {X 0,Y 333.615,Z 352.555,A -85,B 0,C 180,E1 -14442.5,E2 -14442.5} C_VEL
LIN {X 0,Y 333.583,Z 352.558,A -85,B 0,C 180,E1 -14445.956,E2 -14445.956} C_VEL
LIN {X 0,Y 333.592,Z 352.558,A -85,B 0,C 180,E1 -14449.326,E2 -14449.326} C_VEL
LIN {X 0,Y 333.652,Z 352.551,A -85,B 0,C 180,E1 -14453.171,E2 -14453.171} C_VEL
LIN {X 0,Y 333.683,Z 352.661,A -85,B 0,C 180,E1 -14455.711,E2 -14455.711} C_VEL
LIN {X 0,Y 336.395,Z 363.649,A -85,B 0,C 180,E1 -14458.934,E2 -14458.934} C_VEL
LIN {X 0,Y 337.786,Z 369.839,A -85,B 0,C 180,E1 -14460.67,E2 -14460.67} C_VEL
LIN {X 0,Y 345.314,Z 387.797,A -85,B 0,C 180,E1 -14461.789,E2 -14461.789} C_VEL
LIN {X 0,Y 349.475,Z 409.918,A -85,B 0,C 180,E1 -14462.656,E2 -14462.656} C_VEL
LIN {X 0,Y 347.023,Z 507,A -85,B 0,C 180,E1 -14464.672,E2 -14464.672} C_VEL
LIN {X 0,Y 346.082,Z 521.803,A -85,B 0,C 180,E1 -14465.201,E2 -14465.201} C_VEL
LIN {X 0,Y 344.821,Z 535.839,A -85,B 0,C 180,E1 -14465.946,E2 -14465.946} C_VEL
LIN {X 0,Y 343.356,Z 549.758,A -85,B 0,C 180,E1 -14466.957,E2 -14466.957} C_VEL
LIN {X 0,Y 341.761,Z 562.624,A -85,B 0,C 180,E1 -14468.165,E2 -14468.165} C_VEL
LIN {X 0,Y 339.975,Z 574.751,A -85,B 0,C 180,E1 -14469.586,E2 -14469.586} C_VEL
LIN {X 0,Y 338.162,Z 585.928,A -85,B 0,C 180,E1 -14471.21,E2 -14471.21} C_VEL
LIN {X 0,Y 336.5,Z 595.955,A -85,B 0,C 180,E1 -14473.001,E2 -14473.001} C_VEL
LIN {X 0,Y 335.212,Z 604.475,A -85,B 0,C 180,E1 -14474.857,E2 -14474.857} C_VEL
LIN {X 0,Y 334.062,Z 612.247,A -85,B 0,C 180,E1 -14476.931,E2 -14476.931} C_VEL
LIN {X 0,Y 333.061,Z 618.654,A -85,B 0,C 180,E1 -14479.054,E2 -14479.054} C_VEL
LIN {X 0,Y 332.434,Z 624.34,A -85,B 0,C 180,E1 -14481.492,E2 -14481.492} C_VEL
LIN {X 0,Y 332.063,Z 628.749,A -85,B 0,C 180,E1 -14484.121,E2 -14484.121} C_VEL
LIN {X 0,Y 331.949,Z 631.157,A -85,B 0,C 180,E1 -14486.36,E2 -14486.36} C_VEL
LIN {X 0,Y 331.862,Z 632.485,A -85,B 0,C 180,E1 -14488.788,E2 -14488.788} C_VEL
LIN {X 0,Y 331.863,Z 632.479,A -85,B 0,C 180,E1 -14491.215,E2 -14491.215} C_VEL
LIN {X 0,Y 331.95,Z 631.137,A -85,B 0,C 180,E1 -14493.643,E2 -14493.643} C_VEL
LIN {X 0,Y 332.099,Z 628.435,A -85,B 0,C 180,E1 -14496.076,E2 -14496.076} C_VEL
LIN {X 0,Y 332.437,Z 624.301,A -85,B 0,C 180,E1 -14498.512,E2 -14498.512} C_VEL
LIN {X 0,Y 333.065,Z 618.605,A -85,B 0,C 180,E1 -14500.949,E2 -14500.949} C_VEL
LIN {X 0,Y 334.064,Z 612.182,A -85,B 0,C 180,E1 -14503.073,E2 -14503.073} C_VEL
LIN {X 0,Y 335.192,Z 604.463,A -85,B 0,C 180,E1 -14505.13,E2 -14505.13} C_VEL
LIN {X 0,Y 336.514,Z 595.857,A -85,B 0,C 180,E1 -14507.003,E2 -14507.003} C_VEL
LIN {X 0,Y 338.198,Z 585.809,A -85,B 0,C 180,E1 -14508.792,E2 -14508.792} C_VEL
LIN {X 0,Y 339.955,Z 574.597,A -85,B 0,C 180,E1 -14510.419,E2 -14510.419} C_VEL
LIN {X 0,Y 341.739,Z 562.385,A -85,B 0,C 180,E1 -14511.845,E2 -14511.845} C_VEL
LIN {X 0,Y 343.381,Z 549.516,A -85,B 0,C 180,E1 -14513.045,E2 -14513.045} C_VEL
LIN {X 0,Y 344.702,Z 536.67,A -85,B 0,C 180,E1 -14513.987,E2 -14513.987} C_VEL
LIN {X 0,Y 345.999,Z 522.918,A -85,B 0,C 180,E1 -14514.729,E2 -14514.729} C_VEL
LIN {X 0,Y 346.855,Z 508.692,A -85,B 0,C 180,E1 -14515.264,E2 -14515.264} C_VEL
LIN {X 0,Y 347.908,Z 475.053,A -85,B 0,C 180,E1 -14515.985,E2 -14515.985} C_VEL
LIN {X 0,Y 349.369,Z 409.421,A -85,B 0,C 180,E1 -14517.345,E2 -14517.345} C_VEL
LIN {X 0,Y 348.393,Z 403.331,A -85,B 0,C 180,E1 -14517.62,E2 -14517.62} C_VEL
LIN {X 0,Y 348.18,Z 396.961,A -85,B 0,C 180,E1 -14518.107,E2 -14518.107} C_VEL
LIN {X 0,Y 348.418,Z 390.753,A -85,B 0,C 180,E1 -14518.733,E2 -14518.733} C_VEL
LIN {X 0,Y 347.863,Z 387.743,A -85,B 0,C 180,E1 -14519.187,E2 -14519.187} C_VEL
LIN {X 0,Y 345.54,Z 378.984,A -85,B 0,C 180,E1 -14520.816,E2 -14520.816} C_VEL
LIN {X 0,Y 343.086,Z 370.111,A -85,B 0,C 180,E1 -14522.874,E2 -14522.874} C_VEL
LIN {X 0,Y 342.251,Z 367.263,A -85,B 0,C 180,E1 -14523.673,E2 -14523.673} C_VEL
LIN {X 0,Y 339.184,Z 362,A -85,B 0,C 180,E1 -14526.09,E2 -14526.09} C_VEL
LIN {X 0,Y 337.451,Z 359.73,A -85,B 0,C 180,E1 -14527.682,E2 -14527.682} C_VEL
LIN {X 0,Y 336.476,Z 357.369,A -85,B 0,C 180,E1 -14529.392,E2 -14529.392} C_VEL
LIN {X 0,Y 334.97,Z 355.857,A -85,B 0,C 180,E1 -14532.749,E2 -14532.749} C_VEL
LIN {X 0,Y 335.04,Z 356.027,A -85,B 0,C 180,E1 -14535.498,E2 -14535.498} C_VEL
LIN {X 0,Y 336.078,Z 357.046,A -85,B 0,C 180,E1 -14537.996,E2 -14537.996} C_VEL
LIN {X 0,Y 337.837,Z 361.071,A -85,B 0,C 180,E1 -14541.385,E2 -14541.385} C_VEL
LIN {X 0,Y 339.596,Z 365.197,A -85,B 0,C 180,E1 -14543.817,E2 -14543.817} C_VEL
LIN {X 0,Y 341.993,Z 371.663,A -85,B 0,C 180,E1 -14546.776,E2 -14546.776} C_VEL
LIN {X 0,Y 344.076,Z 378.394,A -85,B 0,C 180,E1 -14549.293,E2 -14549.293} C_VEL
LIN {X 0,Y 345.905,Z 386.222,A -85,B 0,C 180,E1 -14551.762,E2 -14551.762} C_VEL
LIN {X 0,Y 349.824,Z 394.198,A -85,B 0,C 180,E1 -14552.922,E2 -14552.922} C_VEL
LIN {X 0,Y 351.386,Z 399.588,A -85,B 0,C 180,E1 -14553.463,E2 -14553.463} C_VEL
LIN {X 0,Y 353.857,Z 411.903,A -85,B 0,C 180,E1 -14554.459,E2 -14554.459} C_VEL
LIN {X 0,Y 350.911,Z 450.307,A -85,B 0,C 180,E1 -14555.799,E2 -14555.799} C_VEL
LIN {X 0,Y 347.583,Z 497.185,A -85,B 0,C 180,E1 -14557.408,E2 -14557.408} C_VEL
LIN {X 0,Y 346.293,Z 511.595,A -85,B 0,C 180,E1 -14558.183,E2 -14558.183} C_VEL
LIN {X 0,Y 344.888,Z 524.194,A -85,B 0,C 180,E1 -14559.108,E2 -14559.108} C_VEL
LIN {X 0,Y 343.221,Z 536.843,A -85,B 0,C 180,E1 -14560.316,E2 -14560.316} C_VEL
LIN {X 0,Y 341.616,Z 546.822,A -85,B 0,C 180,E1 -14561.502,E2 -14561.502} C_VEL
LIN {X 0,Y 340.037,Z 556.196,A -85,B 0,C 180,E1 -14562.871,E2 -14562.871} C_VEL
LIN {X 0,Y 338.436,Z 564.546,A -85,B 0,C 180,E1 -14564.338,E2 -14564.338} C_VEL
LIN {X 0,Y 336.902,Z 572.66,A -85,B 0,C 180,E1 -14566.12,E2 -14566.12} C_VEL
LIN {X 0,Y 335.637,Z 579.206,A -85,B 0,C 180,E1 -14567.913,E2 -14567.913} C_VEL
LIN {X 0,Y 334.518,Z 584.419,A -85,B 0,C 180,E1 -14569.713,E2 -14569.713} C_VEL
LIN {X 0,Y 333.726,Z 588.427,A -85,B 0,C 180,E1 -14571.523,E2 -14571.523} C_VEL
LIN {X 0,Y 333.286,Z 590.48,A -85,B 0,C 180,E1 -14572.731,E2 -14572.731} C_VEL
LIN {X 0,Y 332.805,Z 592.077,A -85,B 0,C 180,E1 -14573.939,E2 -14573.939} C_VEL
LIN {X 0,Y 332.606,Z 593.24,A -85,B 0,C 180,E1 -14575.152,E2 -14575.152} C_VEL
LIN {X 0,Y 332.503,Z 593.946,A -85,B 0,C 180,E1 -14576.365,E2 -14576.365} C_VEL
LIN {X 0,Y 332.332,Z 594.213,A -85,B 0,C 180,E1 -14577.576,E2 -14577.576} C_VEL
LIN {X 0,Y 332.191,Z 594.069,A -85,B 0,C 180,E1 -14578.788,E2 -14578.788} C_VEL
LIN {X 0,Y 332.099,Z 593.484,A -85,B 0,C 180,E1 -14580,E2 -14580} C_VEL
LIN {X 0,Y 332.067,Z 592.43,A -85,B 0,C 180,E1 -14581.213,E2 -14581.213} C_VEL
LIN {X 0,Y 332.086,Z 590.955,A -85,B 0,C 180,E1 -14582.426,E2 -14582.426} C_VEL
LIN {X 0,Y 332.246,Z 587.863,A -85,B 0,C 180,E1 -14584.246,E2 -14584.246} C_VEL
LIN {X 0,Y 332.363,Z 583.645,A -85,B 0,C 180,E1 -14586.069,E2 -14586.069} C_VEL
LIN {X 0,Y 332.643,Z 578.159,A -85,B 0,C 180,E1 -14587.894,E2 -14587.894} C_VEL
LIN {X 0,Y 333.106,Z 571.245,A -85,B 0,C 180,E1 -14589.717,E2 -14589.717} C_VEL
LIN {X 0,Y 333.693,Z 562.653,A -85,B 0,C 180,E1 -14591.542,E2 -14591.542} C_VEL
LIN {X 0,Y 334.381,Z 553.807,A -85,B 0,C 180,E1 -14593.058,E2 -14593.058} C_VEL
LIN {X 0,Y 335.226,Z 543.034,A -85,B 0,C 180,E1 -14594.571,E2 -14594.571} C_VEL
LIN {X 0,Y 335.9,Z 532.346,A -85,B 0,C 180,E1 -14595.783,E2 -14595.783} C_VEL
LIN {X 0,Y 336.557,Z 520.678,A -85,B 0,C 180,E1 -14596.842,E2 -14596.842} C_VEL
LIN {X 0,Y 337.332,Z 507.873,A -85,B 0,C 180,E1 -14597.74,E2 -14597.74} C_VEL
LIN {X 0,Y 337.844,Z 493.689,A -85,B 0,C 180,E1 -14598.457,E2 -14598.457} C_VEL
LIN {X 0,Y 338.389,Z 476.126,A -85,B 0,C 180,E1 -14599.015,E2 -14599.015} C_VEL
LIN {X 0,Y 340.377,Z 404.476,A -85,B 0,C 180,E1 -14601.088,E2 -14601.088} C_VEL
LIN {X 0,Y 336.906,Z 380.175,A -85,B 0,C 180,E1 -14601.973,E2 -14601.973} C_VEL
LIN {X 0,Y 337.276,Z 370.474,A -85,B 0,C 180,E1 -14603.939,E2 -14603.939} C_VEL
LIN {X 0,Y 334.372,Z 355.413,A -85,B 0,C 180,E1 -14607.204,E2 -14607.204} C_VEL
LIN {X 0,Y 333.813,Z 352.531,A -85,B 0,C 180,E1 -14607.88,E2 -14607.88} C_VEL
LIN {X 0,Y 333.639,Z 352.548,A -85,B 0,C 180,E1 -14611.777,E2 -14611.777} C_VEL
LIN {X 0,Y 333.692,Z 352.543,A -85,B 0,C 180,E1 -14614.773,E2 -14614.773} C_VEL
LIN {X 0,Y 333.649,Z 352.551,A -85,B 0,C 180,E1 -14617.652,E2 -14617.652} C_VEL
LIN {X 0,Y 333.609,Z 352.552,A -85,B 0,C 180,E1 -14620.773,E2 -14620.773} C_VEL
LIN {X 0,Y 333.599,Z 352.557,A -85,B 0,C 180,E1 -14624.249,E2 -14624.249} C_VEL
LIN {X 0,Y 333.643,Z 352.553,A -85,B 0,C 180,E1 -14627.617,E2 -14627.617} C_VEL
LIN {X 0,Y 333.639,Z 352.553,A -85,B 0,C 180,E1 -14631.205,E2 -14631.205} C_VEL
LIN {X 0,Y 333.678,Z 352.548,A -85,B 0,C 180,E1 -14633.86,E2 -14633.86} C_VEL
LIN {X 0,Y 333.644,Z 352.605,A -85,B 0,C 180,E1 -14637.067,E2 -14637.067} C_VEL
LIN {X 0,Y 336.348,Z 363.613,A -85,B 0,C 180,E1 -14640.377,E2 -14640.377} C_VEL
LIN {X 0,Y 336.655,Z 364.775,A -85,B 0,C 180,E1 -14640.647,E2 -14640.647} C_VEL
LIN {X 0,Y 345.844,Z 386.055,A -85,B 0,C 180,E1 -14641.994,E2 -14641.994} C_VEL
LIN {X 0,Y 347.598,Z 391.003,A -85,B 0,C 180,E1 -14642.262,E2 -14642.262} C_VEL
LIN {X 0,Y 349.6,Z 402.581,A -85,B 0,C 180,E1 -14642.698,E2 -14642.698} C_VEL
LIN {X 0,Y 347.113,Z 500.074,A -85,B 0,C 180,E1 -14644.716,E2 -14644.716} C_VEL
LIN {X 0,Y 346.411,Z 513.696,A -85,B 0,C 180,E1 -14645.182,E2 -14645.182} C_VEL
LIN {X 0,Y 345.288,Z 526.566,A -85,B 0,C 180,E1 -14645.817,E2 -14645.817} C_VEL
LIN {X 0,Y 344.027,Z 540.018,A -85,B 0,C 180,E1 -14646.73,E2 -14646.73} C_VEL
LIN {X 0,Y 342.512,Z 553.095,A -85,B 0,C 180,E1 -14647.887,E2 -14647.887} C_VEL
LIN {X 0,Y 340.884,Z 564.706,A -85,B 0,C 180,E1 -14649.165,E2 -14649.165} C_VEL
LIN {X 0,Y 339.116,Z 575.616,A -85,B 0,C 180,E1 -14650.633,E2 -14650.633} C_VEL
LIN {X 0,Y 337.674,Z 584.752,A -85,B 0,C 180,E1 -14652.12,E2 -14652.12} C_VEL
LIN {X 0,Y 336.16,Z 593.907,A -85,B 0,C 180,E1 -14653.916,E2 -14653.916} C_VEL
LIN {X 0,Y 334.885,Z 602.646,A -85,B 0,C 180,E1 -14656.033,E2 -14656.033} C_VEL
LIN {X 0,Y 333.779,Z 608.807,A -85,B 0,C 180,E1 -14657.843,E2 -14657.843} C_VEL
LIN {X 0,Y 333.113,Z 613.896,A -85,B 0,C 180,E1 -14659.667,E2 -14659.667} C_VEL
LIN {X 0,Y 332.443,Z 619.17,A -85,B 0,C 180,E1 -14662.1,E2 -14662.1} C_VEL
LIN {X 0,Y 332.222,Z 622.11,A -85,B 0,C 180,E1 -14663.927,E2 -14663.927} C_VEL
LIN {X 0,Y 332.019,Z 624.817,A -85,B 0,C 180,E1 -14666.357,E2 -14666.357} C_VEL
LIN {X 0,Y 331.875,Z 626.176,A -85,B 0,C 180,E1 -14668.785,E2 -14668.785} C_VEL
LIN {X 0,Y 331.875,Z 626.21,A -85,B 0,C 180,E1 -14671.212,E2 -14671.212} C_VEL
LIN {X 0,Y 332.016,Z 624.92,A -85,B 0,C 180,E1 -14673.639,E2 -14673.639} C_VEL
LIN {X 0,Y 332.18,Z 622.274,A -85,B 0,C 180,E1 -14676.071,E2 -14676.071} C_VEL
LIN {X 0,Y 332.57,Z 618.2,A -85,B 0,C 180,E1 -14678.505,E2 -14678.505} C_VEL
LIN {X 0,Y 333.313,Z 612.574,A -85,B 0,C 180,E1 -14680.937,E2 -14680.937} C_VEL
LIN {X 0,Y 334.299,Z 606.225,A -85,B 0,C 180,E1 -14683.06,E2 -14683.06} C_VEL
LIN {X 0,Y 335.339,Z 599.124,A -85,B 0,C 180,E1 -14684.984,E2 -14684.984} C_VEL
LIN {X 0,Y 336.811,Z 590.067,A -85,B 0,C 180,E1 -14686.983,E2 -14686.983} C_VEL
LIN {X 0,Y 338.459,Z 580.113,A -85,B 0,C 180,E1 -14688.773,E2 -14688.773} C_VEL
LIN {X 0,Y 340.254,Z 569.03,A -85,B 0,C 180,E1 -14690.397,E2 -14690.397} C_VEL
LIN {X 0,Y 340.855,Z 564.978,A -85,B 0,C 180,E1 -14690.907,E2 -14690.907} C_VEL
LIN {X 0,Y 340.944,Z 560.286,A -85,B 0,C 180,E1 -14691.512,E2 -14691.512} C_VEL
LIN {X 0,Y 339.349,Z 552.558,A -85,B 0,C 180,E1 -14692.526,E2 -14692.526} C_VEL
LIN {X 0,Y 337.663,Z 544.481,A -85,B 0,C 180,E1 -14693.456,E2 -14693.456} C_VEL
LIN {X 0,Y 337.589,Z 539.247,A -85,B 0,C 180,E1 -14693.92,E2 -14693.92} C_VEL
LIN {X 0,Y 338.965,Z 525.834,A -85,B 0,C 180,E1 -14694.823,E2 -14694.823} C_VEL
LIN {X 0,Y 340.083,Z 511.731,A -85,B 0,C 180,E1 -14695.513,E2 -14695.513} C_VEL
LIN {X 0,Y 340.905,Z 496.81,A -85,B 0,C 180,E1 -14695.979,E2 -14695.979} C_VEL
LIN {X 0,Y 343.324,Z 402.54,A -85,B 0,C 180,E1 -14697.958,E2 -14697.958} C_VEL
LIN {X 0,Y 341.009,Z 391.516,A -85,B 0,C 180,E1 -14698.423,E2 -14698.423} C_VEL
LIN {X 0,Y 333.608,Z 373.986,A -85,B 0,C 180,E1 -14699.539,E2 -14699.539} C_VEL
LIN {X 0,Y 329.283,Z 364.5,A -85,B 0,C 180,E1 -14700.216,E2 -14700.216} C_VEL
LIN {X 0,Y 327.053,Z 355.24,A -85,B 0,C 180,E1 -14703.063,E2 -14703.063} C_VEL
LIN {X 0,Y 326.589,Z 353.433,A -85,B 0,C 180,E1 -14703.656,E2 -14703.656} C_VEL
LIN {X 0,Y 326.616,Z 353.427,A -85,B 0,C 180,E1 -14707.235,E2 -14707.235} C_VEL
LIN {X 0,Y 326.534,Z 353.435,A -85,B 0,C 180,E1 -14711.122,E2 -14711.122} C_VEL
LIN {X 0,Y 326.55,Z 353.433,A -85,B 0,C 180,E1 -14713.524,E2 -14713.524} C_VEL
LIN {X 0,Y 326.564,Z 353.432,A -85,B 0,C 180,E1 -14717.027,E2 -14717.027} C_VEL
LIN {X 0,Y 326.561,Z 353.426,A -85,B 0,C 180,E1 -14720.78,E2 -14720.78} C_VEL
LIN {X 0,Y 326.601,Z 353.428,A -85,B 0,C 180,E1 -14724.479,E2 -14724.479} C_VEL
LIN {X 0,Y 326.595,Z 353.411,A -85,B 0,C 180,E1 -14727.454,E2 -14727.454} C_VEL
LIN {X 0,Y 326.602,Z 353.427,A -85,B 0,C 180,E1 -14730.335,E2 -14730.335} C_VEL
LIN {X 0,Y 326.628,Z 353.406,A -85,B 0,C 180,E1 -14734.644,E2 -14734.644} C_VEL
LIN {X 0,Y 326.601,Z 353.42,A -85,B 0,C 180,E1 -14738.542,E2 -14738.542} C_VEL
LIN {X 0,Y 326.65,Z 353.407,A -85,B 0,C 180,E1 -14742.469,E2 -14742.469} C_VEL
LIN {X 0,Y 326.743,Z 353.406,A -85,B 0,C 180,E1 -14746.314,E2 -14746.314} C_VEL
LIN {X 0,Y 326.769,Z 353.405,A -85,B 0,C 180,E1 -14750.092,E2 -14750.092} C_VEL
LIN {X 0,Y 326.924,Z 353.385,A -85,B 0,C 180,E1 -14753.829,E2 -14753.829} C_VEL
LIN {X 0,Y 326.998,Z 353.376,A -85,B 0,C 180,E1 -14757.536,E2 -14757.536} C_VEL
LIN {X 0,Y 327.033,Z 353.372,A -85,B 0,C 180,E1 -14761.231,E2 -14761.231} C_VEL
LIN {X 0,Y 326.739,Z 353.405,A -85,B 0,C 180,E1 -14763.7,E2 -14763.7} C_VEL
LIN {X 0,Y 326.928,Z 353.386,A -85,B 0,C 180,E1 -14766.17,E2 -14766.17} C_VEL
LIN {X 0,Y 326.766,Z 353.403,A -85,B 0,C 180,E1 -14769.908,E2 -14769.908} C_VEL
LIN {X 0,Y 326.744,Z 353.404,A -85,B 0,C 180,E1 -14773.686,E2 -14773.686} C_VEL
LIN {X 0,Y 326.65,Z 353.416,A -85,B 0,C 180,E1 -14777.531,E2 -14777.531} C_VEL
LIN {X 0,Y 326.6,Z 353.41,A -85,B 0,C 180,E1 -14781.458,E2 -14781.458} C_VEL
LIN {X 0,Y 326.587,Z 353.427,A -85,B 0,C 180,E1 -14785.492,E2 -14785.492} C_VEL
LIN {X 0,Y 326.578,Z 353.414,A -85,B 0,C 180,E1 -14788.258,E2 -14788.258} C_VEL
LIN {X 0,Y 326.559,Z 353.431,A -85,B 0,C 180,E1 -14791.099,E2 -14791.099} C_VEL
LIN {X 0,Y 326.594,Z 353.426,A -85,B 0,C 180,E1 -14794.021,E2 -14794.021} C_VEL
LIN {X 0,Y 326.61,Z 353.426,A -85,B 0,C 180,E1 -14797.238,E2 -14797.238} C_VEL
LIN {X 0,Y 326.531,Z 353.433,A -85,B 0,C 180,E1 -14801.126,E2 -14801.126} C_VEL
LIN {X 0,Y 326.548,Z 353.432,A -85,B 0,C 180,E1 -14803.528,E2 -14803.528} C_VEL
LIN {X 0,Y 326.561,Z 353.434,A -85,B 0,C 180,E1 -14807.031,E2 -14807.031} C_VEL
LIN {X 0,Y 326.562,Z 353.435,A -85,B 0,C 180,E1 -14810.783,E2 -14810.783} C_VEL
LIN {X 0,Y 326.602,Z 353.43,A -85,B 0,C 180,E1 -14814.482,E2 -14814.482} C_VEL
LIN {X 0,Y 326.633,Z 353.432,A -85,B 0,C 180,E1 -14815.1,E2 -14815.1} C_VEL
LIN {X 0,Y 329.466,Z 364.925,A -85,B 0,C 180,E1 -14818.568,E2 -14818.568} C_VEL
LIN {X 0,Y 330.623,Z 370.026,A -85,B 0,C 180,E1 -14819.981,E2 -14819.981} C_VEL
LIN {X 0,Y 338.462,Z 388.305,A -85,B 0,C 180,E1 -14821.178,E2 -14821.178} C_VEL
LIN {X 0,Y 339.609,Z 391.729,A -85,B 0,C 180,E1 -14821.365,E2 -14821.365} C_VEL
LIN {X 0,Y 343.134,Z 410.687,A -85,B 0,C 180,E1 -14822.126,E2 -14822.126} C_VEL
LIN {X 0,Y 340.749,Z 503.976,A -85,B 0,C 180,E1 -14824.09,E2 -14824.09} C_VEL
LIN {X 0,Y 339.891,Z 518.372,A -85,B 0,C 180,E1 -14824.554,E2 -14824.554} C_VEL
LIN {X 0,Y 338.73,Z 532.248,A -85,B 0,C 180,E1 -14825.24,E2 -14825.24} C_VEL
LIN {X 0,Y 337.242,Z 546.156,A -85,B 0,C 180,E1 -14826.188,E2 -14826.188} C_VEL
LIN {X 0,Y 335.757,Z 558.515,A -85,B 0,C 180,E1 -14827.294,E2 -14827.294} C_VEL
LIN {X 0,Y 333.885,Z 571.167,A -85,B 0,C 180,E1 -14828.712,E2 -14828.712} C_VEL
LIN {X 0,Y 332.063,Z 582.018,A -85,B 0,C 180,E1 -14830.209,E2 -14830.209} C_VEL
LIN {X 0,Y 330.252,Z 592.744,A -85,B 0,C 180,E1 -14832.029,E2 -14832.029} C_VEL
LIN {X 0,Y 328.76,Z 601.599,A -85,B 0,C 180,E1 -14833.867,E2 -14833.867} C_VEL
LIN {X 0,Y 327.485,Z 610.088,A -85,B 0,C 180,E1 -14836.031,E2 -14836.031} C_VEL
LIN {X 0,Y 326.301,Z 616.923,A -85,B 0,C 180,E1 -14838.195,E2 -14838.195} C_VEL
LIN {X 0,Y 325.674,Z 621.635,A -85,B 0,C 180,E1 -14840.061,E2 -14840.061} C_VEL
LIN {X 0,Y 325.148,Z 626.523,A -85,B 0,C 180,E1 -14842.55,E2 -14842.55} C_VEL
LIN {X 0,Y 324.889,Z 629.918,A -85,B 0,C 180,E1 -14845.038,E2 -14845.038} C_VEL
LIN {X 0,Y 324.802,Z 631.922,A -85,B 0,C 180,E1 -14847.522,E2 -14847.522} C_VEL
LIN {X 0,Y 324.791,Z 632.582,A -85,B 0,C 180,E1 -14850.002,E2 -14850.002} C_VEL
LIN {X 0,Y 324.802,Z 631.908,A -85,B 0,C 180,E1 -14852.482,E2 -14852.482} C_VEL
LIN {X 0,Y 324.893,Z 629.891,A -85,B 0,C 180,E1 -14854.966,E2 -14854.966} C_VEL
LIN {X 0,Y 325.175,Z 626.485,A -85,B 0,C 180,E1 -14857.453,E2 -14857.453} C_VEL
LIN {X 0,Y 325.678,Z 621.589,A -85,B 0,C 180,E1 -14859.943,E2 -14859.943} C_VEL
LIN {X 0,Y 326.611,Z 615.05,A -85,B 0,C 180,E1 -14862.428,E2 -14862.428} C_VEL
LIN {X 0,Y 327.596,Z 608.893,A -85,B 0,C 180,E1 -14864.285,E2 -14864.285} C_VEL
LIN {X 0,Y 328.748,Z 601.506,A -85,B 0,C 180,E1 -14866.138,E2 -14866.138} C_VEL
LIN {X 0,Y 330.249,Z 592.631,A -85,B 0,C 180,E1 -14867.975,E2 -14867.975} C_VEL
LIN {X 0,Y 332.071,Z 581.883,A -85,B 0,C 180,E1 -14869.795,E2 -14869.795} C_VEL
LIN {X 0,Y 333.863,Z 571.002,A -85,B 0,C 180,E1 -14871.294,E2 -14871.294} C_VEL
LIN {X 0,Y 335.574,Z 559.554,A -85,B 0,C 180,E1 -14872.582,E2 -14872.582} C_VEL
LIN {X 0,Y 337.062,Z 547.677,A -85,B 0,C 180,E1 -14873.666,E2 -14873.666} C_VEL
LIN {X 0,Y 338.365,Z 535.466,A -85,B 0,C 180,E1 -14874.547,E2 -14874.547} C_VEL
LIN {X 0,Y 339.678,Z 521.317,A -85,B 0,C 180,E1 -14875.303,E2 -14875.303} C_VEL
LIN {X 0,Y 340.527,Z 507.471,A -85,B 0,C 180,E1 -14875.809,E2 -14875.809} C_VEL
LIN {X 0,Y 342.497,Z 435.812,A -85,B 0,C 180,E1 -14877.328,E2 -14877.328} C_VEL
LIN {X 0,Y 342.949,Z 420.388,A -85,B 0,C 180,E1 -14877.672,E2 -14877.672} C_VEL
LIN {X 0,Y 343.773,Z 410.189,A -85,B 0,C 180,E1 -14878.08,E2 -14878.08} C_VEL
LIN {X 0,Y 343.045,Z 398.904,A -85,B 0,C 180,E1 -14878.861,E2 -14878.861} C_VEL
LIN {X 0,Y 343.309,Z 393.483,A -85,B 0,C 180,E1 -14879.429,E2 -14879.429} C_VEL
LIN {X 0,Y 340.875,Z 383.472,A -85,B 0,C 180,E1 -14881.299,E2 -14881.299} C_VEL
LIN {X 0,Y 338.504,Z 374.266,A -85,B 0,C 180,E1 -14883.512,E2 -14883.512} C_VEL
LIN {X 0,Y 337.684,Z 372.239,A -85,B 0,C 180,E1 -14884.191,E2 -14884.191} C_VEL
LIN {X 0,Y 335.517,Z 368.456,A -85,B 0,C 180,E1 -14885.911,E2 -14885.911} C_VEL
LIN {X 0,Y 332.966,Z 364.276,A -85,B 0,C 180,E1 -14888.651,E2 -14888.651} C_VEL
LIN {X 0,Y 332.598,Z 363.402,A -85,B 0,C 180,E1 -14889.342,E2 -14889.342} C_VEL
LIN {X 0,Y 331.098,Z 361.895,A -85,B 0,C 180,E1 -14892.019,E2 -14892.019} C_VEL
LIN {X 0,Y 330.739,Z 361.58,A -85,B 0,C 180,E1 -14894.528,E2 -14894.528} C_VEL
LIN {X 0,Y 331.322,Z 362.293,A -85,B 0,C 180,E1 -14897.251,E2 -14897.251} C_VEL
LIN {X 0,Y 331.659,Z 362.577,A -85,B 0,C 180,E1 -14897.875,E2 -14897.875} C_VEL
LIN {X 0,Y 333.148,Z 366.399,A -85,B 0,C 180,E1 -14901.312,E2 -14901.312} C_VEL
LIN {X 0,Y 334.854,Z 370.859,A -85,B 0,C 180,E1 -14904.008,E2 -14904.008} C_VEL
LIN {X 0,Y 336.755,Z 376.317,A -85,B 0,C 180,E1 -14906.596,E2 -14906.596} C_VEL
LIN {X 0,Y 338.697,Z 383.112,A -85,B 0,C 180,E1 -14909.227,E2 -14909.227} C_VEL
LIN {X 0,Y 339.625,Z 386.974,A -85,B 0,C 180,E1 -14910.486,E2 -14910.486} C_VEL
LIN {X 0,Y 344.286,Z 396.013,A -85,B 0,C 180,E1 -14911.998,E2 -14911.998} C_VEL
LIN {X 0,Y 346.003,Z 400.416,A -85,B 0,C 180,E1 -14912.564,E2 -14912.564} C_VEL
LIN {X 0,Y 348.457,Z 412.65,A -85,B 0,C 180,E1 -14913.634,E2 -14913.634} C_VEL
LIN {X 0,Y 348.644,Z 414.807,A -85,B 0,C 180,E1 -14913.776,E2 -14913.776} C_VEL
LIN {X 0,Y 341.856,Z 498.053,A -85,B 0,C 180,E1 -14916.727,E2 -14916.727} C_VEL
LIN {X 0,Y 340.41,Z 512.771,A -85,B 0,C 180,E1 -14917.546,E2 -14917.546} C_VEL
LIN {X 0,Y 338.803,Z 525.906,A -85,B 0,C 180,E1 -14918.555,E2 -14918.555} C_VEL
LIN {X 0,Y 337.091,Z 537.811,A -85,B 0,C 180,E1 -14919.736,E2 -14919.736} C_VEL
LIN {X 0,Y 335.188,Z 548.827,A -85,B 0,C 180,E1 -14921.101,E2 -14921.101} C_VEL
LIN {X 0,Y 333.472,Z 558.112,A -85,B 0,C 180,E1 -14922.523,E2 -14922.523} C_VEL
LIN {X 0,Y 331.519,Z 567.568,A -85,B 0,C 180,E1 -14924.318,E2 -14924.318} C_VEL
LIN {X 0,Y 329.89,Z 575.209,A -85,B 0,C 180,E1 -14926.133,E2 -14926.133} C_VEL
LIN {X 0,Y 328.792,Z 580.383,A -85,B 0,C 180,E1 -14927.658,E2 -14927.658} C_VEL
LIN {X 0,Y 327.605,Z 585.423,A -85,B 0,C 180,E1 -14929.494,E2 -14929.494} C_VEL
LIN {X 0,Y 326.769,Z 589.26,A -85,B 0,C 180,E1 -14931.341,E2 -14931.341} C_VEL
LIN {X 0,Y 326.287,Z 591.2,A -85,B 0,C 180,E1 -14932.575,E2 -14932.575} C_VEL
LIN {X 0,Y 325.785,Z 592.732,A -85,B 0,C 180,E1 -14933.808,E2 -14933.808} C_VEL
LIN {X 0,Y 325.545,Z 593.803,A -85,B 0,C 180,E1 -14935.046,E2 -14935.046} C_VEL
LIN {X 0,Y 325.423,Z 594.405,A -85,B 0,C 180,E1 -14936.285,E2 -14936.285} C_VEL
LIN {X 0,Y 325.248,Z 594.606,A -85,B 0,C 180,E1 -14937.523,E2 -14937.523} C_VEL
LIN {X 0,Y 325.1,Z 594.384,A -85,B 0,C 180,E1 -14938.761,E2 -14938.761} C_VEL
LIN {X 0,Y 325.002,Z 593.684,A -85,B 0,C 180,E1 -14940,E2 -14940} C_VEL
LIN {X 0,Y 324.971,Z 592.564,A -85,B 0,C 180,E1 -14941.239,E2 -14941.239} C_VEL
LIN {X 0,Y 325.035,Z 590.035,A -85,B 0,C 180,E1 -14943.099,E2 -14943.099} C_VEL
LIN {X 0,Y 325.198,Z 586.432,A -85,B 0,C 180,E1 -14944.959,E2 -14944.959} C_VEL
LIN {X 0,Y 325.467,Z 580.817,A -85,B 0,C 180,E1 -14947.101,E2 -14947.101} C_VEL
LIN {X 0,Y 325.802,Z 574.371,A -85,B 0,C 180,E1 -14948.998,E2 -14948.998} C_VEL
LIN {X 0,Y 326.368,Z 566.468,A -85,B 0,C 180,E1 -14950.861,E2 -14950.861} C_VEL
LIN {X 0,Y 327.103,Z 556.527,A -85,B 0,C 180,E1 -14952.723,E2 -14952.723} C_VEL
LIN {X 0,Y 327.887,Z 546.274,A -85,B 0,C 180,E1 -14954.27,E2 -14954.27} C_VEL
LIN {X 0,Y 328.563,Z 536.725,A -85,B 0,C 180,E1 -14955.452,E2 -14955.452} C_VEL
LIN {X 0,Y 329.313,Z 525.52,A -85,B 0,C 180,E1 -14956.585,E2 -14956.585} C_VEL
LIN {X 0,Y 330.017,Z 512.928,A -85,B 0,C 180,E1 -14957.586,E2 -14957.586} C_VEL
LIN {X 0,Y 330.723,Z 498.554,A -85,B 0,C 180,E1 -14958.427,E2 -14958.427} C_VEL
LIN {X 0,Y 331.223,Z 484.794,A -85,B 0,C 180,E1 -14958.96,E2 -14958.96} C_VEL
LIN {X 0,Y 333.47,Z 405.403,A -85,B 0,C 180,E1 -14961.329,E2 -14961.329} C_VEL
LIN {X 0,Y 329.982,Z 380.24,A -85,B 0,C 180,E1 -14962.297,E2 -14962.297} C_VEL
LIN {X 0,Y 330.334,Z 372.68,A -85,B 0,C 180,E1 -14963.843,E2 -14963.843} C_VEL
LIN {X 0,Y 328.547,Z 362.579,A -85,B 0,C 180,E1 -14966.045,E2 -14966.045} C_VEL
LIN {X 0,Y 326.737,Z 353.412,A -85,B 0,C 180,E1 -14968.125,E2 -14968.125} C_VEL
LIN {X 0,Y 326.6,Z 353.423,A -85,B 0,C 180,E1 -14971.094,E2 -14971.094} C_VEL
LIN {X 0,Y 326.613,Z 353.425,A -85,B 0,C 180,E1 -14974.019,E2 -14974.019} C_VEL
LIN {X 0,Y 326.629,Z 353.423,A -85,B 0,C 180,E1 -14977.237,E2 -14977.237} C_VEL
LIN {X 0,Y 326.55,Z 353.432,A -85,B 0,C 180,E1 -14981.124,E2 -14981.124} C_VEL
LIN {X 0,Y 326.567,Z 353.432,A -85,B 0,C 180,E1 -14983.525,E2 -14983.525} C_VEL
LIN {X 0,Y 326.579,Z 353.43,A -85,B 0,C 180,E1 -14987.028,E2 -14987.028} C_VEL
LIN {X 0,Y 326.587,Z 353.431,A -85,B 0,C 180,E1 -14991.384,E2 -14991.384} C_VEL
LIN {X 0,Y 326.623,Z 353.42,A -85,B 0,C 180,E1 -14994.851,E2 -14994.851} C_VEL
LIN {X 0,Y 326.607,Z 353.504,A -85,B 0,C 180,E1 -14996.502,E2 -14996.502} C_VEL
LIN {X 0,Y 329.374,Z 364.589,A -85,B 0,C 180,E1 -14999.925,E2 -14999.925} C_VEL
LIN {X 0,Y 338.999,Z 386.488,A -85,B 0,C 180,E1 -15001.385,E2 -15001.385} C_VEL
LIN {X 0,Y 341.543,Z 393.352,A -85,B 0,C 180,E1 -15001.779,E2 -15001.779} C_VEL
LIN {X 0,Y 343.276,Z 402.753,A -85,B 0,C 180,E1 -15002.153,E2 -15002.153} C_VEL
LIN {X 0,Y 340.787,Z 498.657,A -85,B 0,C 180,E1 -15004.171,E2 -15004.171} C_VEL
LIN {X 0,Y 340.136,Z 511.032,A -85,B 0,C 180,E1 -15004.57,E2 -15004.57} C_VEL
LIN {X 0,Y 338.941,Z 525.343,A -85,B 0,C 180,E1 -15005.253,E2 -15005.253} C_VEL
LIN {X 0,Y 337.69,Z 538.323,A -85,B 0,C 180,E1 -15006.12,E2 -15006.12} C_VEL
LIN {X 0,Y 336.23,Z 550.801,A -85,B 0,C 180,E1 -15007.197,E2 -15007.197} C_VEL
LIN {X 0,Y 334.457,Z 563.598,A -85,B 0,C 180,E1 -15008.584,E2 -15008.584} C_VEL
LIN {X 0,Y 332.783,Z 573.692,A -85,B 0,C 180,E1 -15009.928,E2 -15009.928} C_VEL
LIN {X 0,Y 331.215,Z 583.111,A -85,B 0,C 180,E1 -15011.439,E2 -15011.439} C_VEL
LIN {X 0,Y 329.557,Z 592.577,A -85,B 0,C 180,E1 -15013.266,E2 -15013.266} C_VEL
LIN {X 0,Y 328.304,Z 600.417,A -85,B 0,C 180,E1 -15015.113,E2 -15015.113} C_VEL
LIN {X 0,Y 327.2,Z 606.941,A -85,B 0,C 180,E1 -15016.964,E2 -15016.964} C_VEL
LIN {X 0,Y 326.334,Z 612.357,A -85,B 0,C 180,E1 -15018.822,E2 -15018.822} C_VEL
LIN {X 0,Y 325.526,Z 618.047,A -85,B 0,C 180,E1 -15021.306,E2 -15021.306} C_VEL
LIN {X 0,Y 325.146,Z 622.293,A -85,B 0,C 180,E1 -15023.874,E2 -15023.874} C_VEL
LIN {X 0,Y 324.928,Z 624.885,A -85,B 0,C 180,E1 -15026.278,E2 -15026.278} C_VEL
LIN {X 0,Y 324.787,Z 626.243,A -85,B 0,C 180,E1 -15028.758,E2 -15028.758} C_VEL
LIN {X 0,Y 324.786,Z 626.277,A -85,B 0,C 180,E1 -15031.238,E2 -15031.238} C_VEL
LIN {X 0,Y 324.925,Z 624.987,A -85,B 0,C 180,E1 -15033.719,E2 -15033.719} C_VEL
LIN {X 0,Y 325.11,Z 622.341,A -85,B 0,C 180,E1 -15036.203,E2 -15036.203} C_VEL
LIN {X 0,Y 325.521,Z 618.267,A -85,B 0,C 180,E1 -15038.69,E2 -15038.69} C_VEL
LIN {X 0,Y 326.306,Z 612.64,A -85,B 0,C 180,E1 -15041.175,E2 -15041.175} C_VEL
LIN {X 0,Y 327.363,Z 606.291,A -85,B 0,C 180,E1 -15043.341,E2 -15043.341} C_VEL
LIN {X 0,Y 328.408,Z 599.434,A -85,B 0,C 180,E1 -15045.245,E2 -15045.245} C_VEL
LIN {X 0,Y 330.001,Z 590.132,A -85,B 0,C 180,E1 -15047.345,E2 -15047.345} C_VEL
LIN {X 0,Y 331.725,Z 580.178,A -85,B 0,C 180,E1 -15049.169,E2 -15049.169} C_VEL
LIN {X 0,Y 333.594,Z 569.094,A -85,B 0,C 180,E1 -15050.823,E2 -15050.823} C_VEL
LIN {X 0,Y 335.299,Z 558.062,A -85,B 0,C 180,E1 -15052.164,E2 -15052.164} C_VEL
LIN {X 0,Y 336.898,Z 545.737,A -85,B 0,C 180,E1 -15053.381,E2 -15053.381} C_VEL
LIN {X 0,Y 337.589,Z 539.247,A -85,B 0,C 180,E1 -15053.92,E2 -15053.92} C_VEL
LIN {X 0,Y 337.574,Z 533.908,A -85,B 0,C 180,E1 -15054.36,E2 -15054.36} C_VEL
LIN {X 0,Y 335.802,Z 525.208,A -85,B 0,C 180,E1 -15055.115,E2 -15055.115} C_VEL
LIN {X 0,Y 334.007,Z 516.316,A -85,B 0,C 180,E1 -15055.789,E2 -15055.789} C_VEL
LIN {X 0,Y 333.78,Z 510.681,A -85,B 0,C 180,E1 -15056.081,E2 -15056.081} C_VEL
LIN {X 0,Y 334.535,Z 496.857,A -85,B 0,C 180,E1 -15056.512,E2 -15056.512} C_VEL
LIN {X 0,Y 337.058,Z 404.668,A -85,B 0,C 180,E1 -15058.475,E2 -15058.475} C_VEL
LIN {X 0,Y 335.434,Z 395.186,A -85,B 0,C 180,E1 -15058.853,E2 -15058.853} C_VEL
LIN {X 0,Y 329.042,Z 379.699,A -85,B 0,C 180,E1 -15059.85,E2 -15059.85} C_VEL
LIN {X 0,Y 322.094,Z 364.542,A -85,B 0,C 180,E1 -15060.973,E2 -15060.973} C_VEL
LIN {X 0,Y 319.581,Z 354.307,A -85,B 0,C 180,E1 -15064.297,E2 -15064.297} C_VEL
LIN {X 0,Y 319.525,Z 354.309,A -85,B 0,C 180,E1 -15068.012,E2 -15068.012} C_VEL
LIN {X 0,Y 319.495,Z 354.312,A -85,B 0,C 180,E1 -15071.59,E2 -15071.59} C_VEL
LIN {X 0,Y 319.477,Z 354.313,A -85,B 0,C 180,E1 -15074.741,E2 -15074.741} C_VEL
LIN {X 0,Y 319.542,Z 354.307,A -85,B 0,C 180,E1 -15077.014,E2 -15077.014} C_VEL
LIN {X 0,Y 319.504,Z 354.312,A -85,B 0,C 180,E1 -15080.364,E2 -15080.364} C_VEL
LIN {X 0,Y 319.569,Z 354.303,A -85,B 0,C 180,E1 -15084.456,E2 -15084.456} C_VEL
LIN {X 0,Y 319.511,Z 354.296,A -85,B 0,C 180,E1 -15088.136,E2 -15088.136} C_VEL
LIN {X 0,Y 319.556,Z 354.299,A -85,B 0,C 180,E1 -15091.603,E2 -15091.603} C_VEL
LIN {X 0,Y 319.559,Z 354.296,A -85,B 0,C 180,E1 -15095.3,E2 -15095.3} C_VEL
LIN {X 0,Y 319.551,Z 354.304,A -85,B 0,C 180,E1 -15098.044,E2 -15098.044} C_VEL
LIN {X 0,Y 319.6,Z 354.282,A -85,B 0,C 180,E1 -15102.07,E2 -15102.07} C_VEL
LIN {X 0,Y 319.717,Z 354.282,A -85,B 0,C 180,E1 -15106.007,E2 -15106.007} C_VEL
LIN {X 0,Y 319.721,Z 354.282,A -85,B 0,C 180,E1 -15109.872,E2 -15109.872} C_VEL
LIN {X 0,Y 319.881,Z 354.262,A -85,B 0,C 180,E1 -15113.693,E2 -15113.693} C_VEL
LIN {X 0,Y 319.945,Z 354.255,A -85,B 0,C 180,E1 -15117.482,E2 -15117.482} C_VEL
LIN {X 0,Y 320,Z 354.248,A -85,B 0,C 180,E1 -15121.258,E2 -15121.258} C_VEL
LIN {X 0,Y 319.705,Z 354.284,A -85,B 0,C 180,E1 -15125.045,E2 -15125.045} C_VEL
LIN {X 0,Y 319.838,Z 354.266,A -85,B 0,C 180,E1 -15127.576,E2 -15127.576} C_VEL
LIN {X 0,Y 319.697,Z 354.285,A -85,B 0,C 180,E1 -15131.411,E2 -15131.411} C_VEL
LIN {X 0,Y 319.699,Z 354.288,A -85,B 0,C 180,E1 -15134.712,E2 -15134.712} C_VEL
LIN {X 0,Y 319.6,Z 354.295,A -85,B 0,C 180,E1 -15137.93,E2 -15137.93} C_VEL
LIN {X 0,Y 319.551,Z 354.284,A -85,B 0,C 180,E1 -15141.956,E2 -15141.956} C_VEL
LIN {X 0,Y 319.536,Z 354.309,A -85,B 0,C 180,E1 -15146.097,E2 -15146.097} C_VEL
LIN {X 0,Y 319.512,Z 354.291,A -85,B 0,C 180,E1 -15148.941,E2 -15148.941} C_VEL
LIN {X 0,Y 319.511,Z 354.31,A -85,B 0,C 180,E1 -15151.864,E2 -15151.864} C_VEL
LIN {X 0,Y 319.566,Z 354.302,A -85,B 0,C 180,E1 -15155.544,E2 -15155.544} C_VEL
LIN {X 0,Y 319.517,Z 354.31,A -85,B 0,C 180,E1 -15159.663,E2 -15159.663} C_VEL
LIN {X 0,Y 319.508,Z 354.309,A -85,B 0,C 180,E1 -15163.461,E2 -15163.461} C_VEL
LIN {X 0,Y 319.54,Z 354.309,A -85,B 0,C 180,E1 -15167.017,E2 -15167.017} C_VEL
LIN {X 0,Y 319.505,Z 354.315,A -85,B 0,C 180,E1 -15170.368,E2 -15170.368} C_VEL
LIN {X 0,Y 319.574,Z 354.305,A -85,B 0,C 180,E1 -15174.459,E2 -15174.459} C_VEL
LIN {X 0,Y 322.101,Z 364.536,A -85,B 0,C 180,E1 -15177.676,E2 -15177.676} C_VEL
LIN {X 0,Y 323.32,Z 369.714,A -85,B 0,C 180,E1 -15179.224,E2 -15179.224} C_VEL
LIN {X 0,Y 332.138,Z 389.849,A -85,B 0,C 180,E1 -15180.615,E2 -15180.615} C_VEL
LIN {X 0,Y 333.666,Z 394.274,A -85,B 0,C 180,E1 -15180.869,E2 -15180.869} C_VEL
LIN {X 0,Y 336.866,Z 412.544,A -85,B 0,C 180,E1 -15181.606,E2 -15181.606} C_VEL
LIN {X 0,Y 334.246,Z 506.896,A -85,B 0,C 180,E1 -15183.631,E2 -15183.631} C_VEL
LIN {X 0,Y 333.237,Z 521.686,A -85,B 0,C 180,E1 -15184.176,E2 -15184.176} C_VEL
LIN {X 0,Y 331.925,Z 535.718,A -85,B 0,C 180,E1 -15184.948,E2 -15184.948} C_VEL
LIN {X 0,Y 330.307,Z 549.633,A -85,B 0,C 180,E1 -15185.99,E2 -15185.99} C_VEL
LIN {X 0,Y 328.653,Z 561.893,A -85,B 0,C 180,E1 -15187.176,E2 -15187.176} C_VEL
LIN {X 0,Y 326.858,Z 573.452,A -85,B 0,C 180,E1 -15188.562,E2 -15188.562} C_VEL
LIN {X 0,Y 325.04,Z 583.907,A -85,B 0,C 180,E1 -15190.092,E2 -15190.092} C_VEL
LIN {X 0,Y 323.179,Z 594.307,A -85,B 0,C 180,E1 -15191.95,E2 -15191.95} C_VEL
LIN {X 0,Y 321.647,Z 603.012,A -85,B 0,C 180,E1 -15193.856,E2 -15193.856} C_VEL
LIN {X 0,Y 320.361,Z 611.105,A -85,B 0,C 180,E1 -15196.038,E2 -15196.038} C_VEL
LIN {X 0,Y 319.337,Z 616.856,A -85,B 0,C 180,E1 -15197.934,E2 -15197.934} C_VEL
LIN {X 0,Y 318.629,Z 621.568,A -85,B 0,C 180,E1 -15199.839,E2 -15199.839} C_VEL
LIN {X 0,Y 318.072,Z 626.456,A -85,B 0,C 180,E1 -15202.384,E2 -15202.384} C_VEL
LIN {X 0,Y 317.809,Z 629.852,A -85,B 0,C 180,E1 -15204.927,E2 -15204.927} C_VEL
LIN {X 0,Y 317.725,Z 631.855,A -85,B 0,C 180,E1 -15207.466,E2 -15207.466} C_VEL
LIN {X 0,Y 317.702,Z 632.514,A -85,B 0,C 180,E1 -15210.002,E2 -15210.002} C_VEL
LIN {X 0,Y 317.725,Z 631.841,A -85,B 0,C 180,E1 -15212.537,E2 -15212.537} C_VEL
LIN {X 0,Y 317.814,Z 629.823,A -85,B 0,C 180,E1 -15215.077,E2 -15215.077} C_VEL
LIN {X 0,Y 318.094,Z 626.417,A -85,B 0,C 180,E1 -15217.62,E2 -15217.62} C_VEL
LIN {X 0,Y 318.633,Z 621.52,A -85,B 0,C 180,E1 -15220.165,E2 -15220.165} C_VEL
LIN {X 0,Y 319.34,Z 616.795,A -85,B 0,C 180,E1 -15222.07,E2 -15222.07} C_VEL
LIN {X 0,Y 320.535,Z 609.942,A -85,B 0,C 180,E1 -15224.282,E2 -15224.282} C_VEL
LIN {X 0,Y 321.879,Z 601.437,A -85,B 0,C 180,E1 -15226.492,E2 -15226.492} C_VEL
LIN {X 0,Y 323.477,Z 592.561,A -85,B 0,C 180,E1 -15228.365,E2 -15228.365} C_VEL
LIN {X 0,Y 325.359,Z 581.812,A -85,B 0,C 180,E1 -15230.221,E2 -15230.221} C_VEL
LIN {X 0,Y 327.252,Z 570.931,A -85,B 0,C 180,E1 -15231.746,E2 -15231.746} C_VEL
LIN {X 0,Y 329.141,Z 558.674,A -85,B 0,C 180,E1 -15233.142,E2 -15233.142} C_VEL
LIN {X 0,Y 330.762,Z 545.823,A -85,B 0,C 180,E1 -15234.312,E2 -15234.312} C_VEL
LIN {X 0,Y 332.181,Z 533.104,A -85,B 0,C 180,E1 -15235.202,E2 -15235.202} C_VEL
LIN {X 0,Y 333.451,Z 518.693,A -85,B 0,C 180,E1 -15235.936,E2 -15235.936} C_VEL
LIN {X 0,Y 334.261,Z 504.528,A -85,B 0,C 180,E1 -15236.414,E2 -15236.414} C_VEL
LIN {X 0,Y 335.939,Z 445.208,A -85,B 0,C 180,E1 -15237.683,E2 -15237.683} C_VEL
LIN {X 0,Y 336.335,Z 438.383,A -85,B 0,C 180,E1 -15237.886,E2 -15237.886} C_VEL
LIN {X 0,Y 338.98,Z 412.097,A -85,B 0,C 180,E1 -15238.896,E2 -15238.896} C_VEL
LIN {X 0,Y 338.198,Z 398.223,A -85,B 0,C 180,E1 -15239.918,E2 -15239.918} C_VEL
LIN {X 0,Y 338.255,Z 396.732,A -85,B 0,C 180,E1 -15240.097,E2 -15240.097} C_VEL
LIN {X 0,Y 336.221,Z 387.96,A -85,B 0,C 180,E1 -15241.802,E2 -15241.802} C_VEL
LIN {X 0,Y 334.071,Z 378.965,A -85,B 0,C 180,E1 -15244.017,E2 -15244.017} C_VEL
LIN {X 0,Y 331.275,Z 373.926,A -85,B 0,C 180,E1 -15246.277,E2 -15246.277} C_VEL
LIN {X 0,Y 329.335,Z 370.948,A -85,B 0,C 180,E1 -15248.235,E2 -15248.235} C_VEL
LIN {X 0,Y 328.198,Z 368.885,A -85,B 0,C 180,E1 -15249.974,E2 -15249.974} C_VEL
LIN {X 0,Y 326.817,Z 367.441,A -85,B 0,C 180,E1 -15253.017,E2 -15253.017} C_VEL
LIN {X 0,Y 326.61,Z 367.393,A -85,B 0,C 180,E1 -15255.245,E2 -15255.245} C_VEL
LIN {X 0,Y 326.94,Z 367.825,A -85,B 0,C 180,E1 -15256.962,E2 -15256.962} C_VEL
LIN {X 0,Y 327.411,Z 369.015,A -85,B 0,C 180,E1 -15258.704,E2 -15258.704} C_VEL
LIN {X 0,Y 328.675,Z 372.386,A -85,B 0,C 180,E1 -15261.676,E2 -15261.676} C_VEL
LIN {X 0,Y 330.009,Z 376.195,A -85,B 0,C 180,E1 -15264.026,E2 -15264.026} C_VEL
LIN {X 0,Y 331.979,Z 382.417,A -85,B 0,C 180,E1 -15267.008,E2 -15267.008} C_VEL
LIN {X 0,Y 333.388,Z 387.666,A -85,B 0,C 180,E1 -15269.024,E2 -15269.024} C_VEL
LIN {X 0,Y 337.724,Z 395.74,A -85,B 0,C 180,E1 -15270.62,E2 -15270.62} C_VEL
LIN {X 0,Y 341.029,Z 402.768,A -85,B 0,C 180,E1 -15271.744,E2 -15271.744} C_VEL
LIN {X 0,Y 342.851,Z 411.358,A -85,B 0,C 180,E1 -15272.583,E2 -15272.583} C_VEL
LIN {X 0,Y 343.576,Z 415.923,A -85,B 0,C 180,E1 -15272.963,E2 -15272.963} C_VEL
LIN {X 0,Y 336.287,Z 498.587,A -85,B 0,C 180,E1 -15275.991,E2 -15275.991} C_VEL
LIN {X 0,Y 334.751,Z 513.124,A -85,B 0,C 180,E1 -15276.818,E2 -15276.818} C_VEL
LIN {X 0,Y 333.019,Z 526.174,A -85,B 0,C 180,E1 -15277.838,E2 -15277.838} C_VEL
LIN {X 0,Y 331.091,Z 538.556,A -85,B 0,C 180,E1 -15279.091,E2 -15279.091} C_VEL
LIN {X 0,Y 328.99,Z 549.862,A -85,B 0,C 180,E1 -15280.53,E2 -15280.53} C_VEL
LIN {X 0,Y 326.922,Z 560.034,A -85,B 0,C 180,E1 -15282.161,E2 -15282.161} C_VEL
LIN {X 0,Y 324.896,Z 569.206,A -85,B 0,C 180,E1 -15283.99,E2 -15283.99} C_VEL
LIN {X 0,Y 323.152,Z 576.549,A -85,B 0,C 180,E1 -15285.838,E2 -15285.838} C_VEL
LIN {X 0,Y 321.52,Z 583.321,A -85,B 0,C 180,E1 -15288.015,E2 -15288.015} C_VEL
LIN {X 0,Y 320.387,Z 587.778,A -85,B 0,C 180,E1 -15289.893,E2 -15289.893} C_VEL
LIN {X 0,Y 319.548,Z 591.091,A -85,B 0,C 180,E1 -15291.782,E2 -15291.782} C_VEL
LIN {X 0,Y 318.768,Z 593.393,A -85,B 0,C 180,E1 -15293.671,E2 -15293.671} C_VEL
LIN {X 0,Y 318.488,Z 594.339,A -85,B 0,C 180,E1 -15294.936,E2 -15294.936} C_VEL
LIN {X 0,Y 318.345,Z 594.87,A -85,B 0,C 180,E1 -15296.203,E2 -15296.203} C_VEL
LIN {X 0,Y 318.164,Z 594.997,A -85,B 0,C 180,E1 -15297.468,E2 -15297.468} C_VEL
LIN {X 0,Y 318.007,Z 594.649,A -85,B 0,C 180,E1 -15298.734,E2 -15298.734} C_VEL
LIN {X 0,Y 317.905,Z 593.875,A -85,B 0,C 180,E1 -15300,E2 -15300} C_VEL
LIN {X 0,Y 317.877,Z 592.684,A -85,B 0,C 180,E1 -15301.267,E2 -15301.267} C_VEL
LIN {X 0,Y 317.96,Z 590.012,A -85,B 0,C 180,E1 -15303.168,E2 -15303.168} C_VEL
LIN {X 0,Y 318.1,Z 586.254,A -85,B 0,C 180,E1 -15305.07,E2 -15305.07} C_VEL
LIN {X 0,Y 318.375,Z 580.994,A -85,B 0,C 180,E1 -15307.071,E2 -15307.071} C_VEL
LIN {X 0,Y 318.75,Z 573.807,A -85,B 0,C 180,E1 -15309.198,E2 -15309.198} C_VEL
LIN {X 0,Y 319.359,Z 565.61,A -85,B 0,C 180,E1 -15311.102,E2 -15311.102} C_VEL
LIN {X 0,Y 319.964,Z 557.246,A -85,B 0,C 180,E1 -15312.689,E2 -15312.689} C_VEL
LIN {X 0,Y 320.742,Z 547.101,A -85,B 0,C 180,E1 -15314.271,E2 -15314.271} C_VEL
LIN {X 0,Y 321.516,Z 536.838,A -85,B 0,C 180,E1 -15315.571,E2 -15315.571} C_VEL
LIN {X 0,Y 322.321,Z 524.933,A -85,B 0,C 180,E1 -15316.793,E2 -15316.793} C_VEL
LIN {X 0,Y 322.994,Z 513.194,A -85,B 0,C 180,E1 -15317.736,E2 -15317.736} C_VEL
LIN {X 0,Y 323.698,Z 498.88,A -85,B 0,C 180,E1 -15318.596,E2 -15318.596} C_VEL
LIN {X 0,Y 324.211,Z 485.28,A -85,B 0,C 180,E1 -15319.14,E2 -15319.14} C_VEL
LIN {X 0,Y 326.517,Z 406.056,A -85,B 0,C 180,E1 -15321.581,E2 -15321.581} C_VEL
LIN {X 0,Y 323.049,Z 380.612,A -85,B 0,C 180,E1 -15322.566,E2 -15322.566} C_VEL
LIN {X 0,Y 323.321,Z 373.313,A -85,B 0,C 180,E1 -15324.081,E2 -15324.081} C_VEL
LIN {X 0,Y 320.783,Z 359.719,A -85,B 0,C 180,E1 -15327.089,E2 -15327.089} C_VEL
LIN {X 0,Y 319.691,Z 354.29,A -85,B 0,C 180,E1 -15328.306,E2 -15328.306} C_VEL
LIN {X 0,Y 319.539,Z 354.305,A -85,B 0,C 180,E1 -15331.861,E2 -15331.861} C_VEL
LIN {X 0,Y 319.586,Z 354.302,A -85,B 0,C 180,E1 -15335.542,E2 -15335.542} C_VEL
LIN {X 0,Y 319.534,Z 354.309,A -85,B 0,C 180,E1 -15339.661,E2 -15339.661} C_VEL
LIN {X 0,Y 319.526,Z 354.309,A -85,B 0,C 180,E1 -15343.459,E2 -15343.459} C_VEL
LIN {X 0,Y 319.558,Z 354.305,A -85,B 0,C 180,E1 -15347.015,E2 -15347.015} C_VEL
LIN {X 0,Y 319.551,Z 354.305,A -85,B 0,C 180,E1 -15350.37,E2 -15350.37} C_VEL
LIN {X 0,Y 319.583,Z 354.3,A -85,B 0,C 180,E1 -15354.457,E2 -15354.457} C_VEL
LIN {X 0,Y 319.572,Z 354.335,A -85,B 0,C 180,E1 -15355.888,E2 -15355.888} C_VEL
LIN {X 0,Y 322.156,Z 364.663,A -85,B 0,C 180,E1 -15359.177,E2 -15359.177} C_VEL
LIN {X 0,Y 330.753,Z 383.739,A -85,B 0,C 180,E1 -15360.533,E2 -15360.533} C_VEL
LIN {X 0,Y 335.498,Z 395.596,A -85,B 0,C 180,E1 -15361.275,E2 -15361.275} C_VEL
LIN {X 0,Y 336.99,Z 403.663,A -85,B 0,C 180,E1 -15361.607,E2 -15361.607} C_VEL
LIN {X 0,Y 334.616,Z 492.34,A -85,B 0,C 180,E1 -15363.491,E2 -15363.491} C_VEL
LIN {X 0,Y 333.94,Z 507.332,A -85,B 0,C 180,E1 -15363.895,E2 -15363.895} C_VEL
LIN {X 0,Y 333.014,Z 520.068,A -85,B 0,C 180,E1 -15364.447,E2 -15364.447} C_VEL
LIN {X 0,Y 331.728,Z 533.595,A -85,B 0,C 180,E1 -15365.263,E2 -15365.263} C_VEL
LIN {X 0,Y 330.222,Z 546.65,A -85,B 0,C 180,E1 -15366.313,E2 -15366.313} C_VEL
LIN {X 0,Y 328.595,Z 558.527,A -85,B 0,C 180,E1 -15367.521,E2 -15367.521} C_VEL
LIN {X 0,Y 326.651,Z 570.56,A -85,B 0,C 180,E1 -15369.04,E2 -15369.04} C_VEL
LIN {X 0,Y 324.794,Z 581.403,A -85,B 0,C 180,E1 -15370.73,E2 -15370.73} C_VEL
LIN {X 0,Y 322.972,Z 591.165,A -85,B 0,C 180,E1 -15372.588,E2 -15372.588} C_VEL
LIN {X 0,Y 321.603,Z 599.116,A -85,B 0,C 180,E1 -15374.433,E2 -15374.433} C_VEL
LIN {X 0,Y 320.478,Z 606.005,A -85,B 0,C 180,E1 -15376.363,E2 -15376.363} C_VEL
LIN {X 0,Y 319.342,Z 612.426,A -85,B 0,C 180,E1 -15378.574,E2 -15378.574} C_VEL
LIN {X 0,Y 318.496,Z 618.115,A -85,B 0,C 180,E1 -15381.113,E2 -15381.113} C_VEL
LIN {X 0,Y 318.07,Z 622.247,A -85,B 0,C 180,E1 -15383.655,E2 -15383.655} C_VEL
LIN {X 0,Y 317.84,Z 624.953,A -85,B 0,C 180,E1 -15386.195,E2 -15386.195} C_VEL
LIN {X 0,Y 317.701,Z 626.311,A -85,B 0,C 180,E1 -15388.731,E2 -15388.731} C_VEL
LIN {X 0,Y 317.701,Z 626.344,A -85,B 0,C 180,E1 -15391.266,E2 -15391.266} C_VEL
LIN {X 0,Y 317.836,Z 625.054,A -85,B 0,C 180,E1 -15393.802,E2 -15393.802} C_VEL
LIN {X 0,Y 318.053,Z 622.408,A -85,B 0,C 180,E1 -15396.341,E2 -15396.341} C_VEL
LIN {X 0,Y 318.487,Z 618.333,A -85,B 0,C 180,E1 -15398.884,E2 -15398.884} C_VEL
LIN {X 0,Y 319.315,Z 612.706,A -85,B 0,C 180,E1 -15401.423,E2 -15401.423} C_VEL
LIN {X 0,Y 320.423,Z 606.356,A -85,B 0,C 180,E1 -15403.636,E2 -15403.636} C_VEL
LIN {X 0,Y 321.697,Z 598.573,A -85,B 0,C 180,E1 -15405.816,E2 -15405.816} C_VEL
LIN {X 0,Y 323.21,Z 590.197,A -85,B 0,C 180,E1 -15407.721,E2 -15407.721} C_VEL
LIN {X 0,Y 325.006,Z 580.242,A -85,B 0,C 180,E1 -15409.581,E2 -15409.581} C_VEL
LIN {X 0,Y 326.925,Z 569.157,A -85,B 0,C 180,E1 -15411.268,E2 -15411.268} C_VEL
LIN {X 0,Y 328.908,Z 557.111,A -85,B 0,C 180,E1 -15412.738,E2 -15412.738} C_VEL
LIN {X 0,Y 330.544,Z 544.39,A -85,B 0,C 180,E1 -15413.991,E2 -15413.991} C_VEL
LIN {X 0,Y 331.962,Z 531.755,A -85,B 0,C 180,E1 -15414.965,E2 -15414.965} C_VEL
LIN {X 0,Y 333.272,Z 517.579,A -85,B 0,C 180,E1 -15415.779,E2 -15415.779} C_VEL
LIN {X 0,Y 333.78,Z 510.681,A -85,B 0,C 180,E1 -15416.081,E2 -15416.081} C_VEL
LIN {X 0,Y 333.542,Z 504.971,A -85,B 0,C 180,E1 -15416.339,E2 -15416.339} C_VEL
LIN {X 0,Y 329.111,Z 486.365,A -85,B 0,C 180,E1 -15417.25,E2 -15417.25} C_VEL
LIN {X 0,Y 328.709,Z 480.555,A -85,B 0,C 180,E1 -15417.423,E2 -15417.423} C_VEL
LIN {X 0,Y 330.818,Z 405.077,A -85,B 0,C 180,E1 -15419.054,E2 -15419.054} C_VEL
LIN {X 0,Y 329.179,Z 396.896,A -85,B 0,C 180,E1 -15419.414,E2 -15419.414} C_VEL
LIN {X 0,Y 321.371,Z 378.349,A -85,B 0,C 180,E1 -15420.674,E2 -15420.674} C_VEL
LIN {X 0,Y 314.857,Z 364.608,A -85,B 0,C 180,E1 -15421.769,E2 -15421.769} C_VEL
LIN {X 0,Y 312.529,Z 355.183,A -85,B 0,C 180,E1 -15424.889,E2 -15424.889} C_VEL
LIN {X 0,Y 312.476,Z 355.187,A -85,B 0,C 180,E1 -15428.075,E2 -15428.075} C_VEL
LIN {X 0,Y 312.445,Z 355.19,A -85,B 0,C 180,E1 -15432.073,E2 -15432.073} C_VEL
LIN {X 0,Y 312.448,Z 355.189,A -85,B 0,C 180,E1 -15436.033,E2 -15436.033} C_VEL
LIN {X 0,Y 312.445,Z 355.19,A -85,B 0,C 180,E1 -15439.884,E2 -15439.884} C_VEL
LIN {X 0,Y 312.523,Z 355.179,A -85,B 0,C 180,E1 -15444.049,E2 -15444.049} C_VEL
LIN {X 0,Y 312.489,Z 355.167,A -85,B 0,C 180,E1 -15447.332,E2 -15447.332} C_VEL
LIN {X 0,Y 312.492,Z 355.18,A -85,B 0,C 180,E1 -15451.291,E2 -15451.291} C_VEL
LIN {X 0,Y 312.533,Z 355.162,A -85,B 0,C 180,E1 -15454.706,E2 -15454.706} C_VEL
LIN {X 0,Y 312.509,Z 355.171,A -85,B 0,C 180,E1 -15458.911,E2 -15458.911} C_VEL
LIN {X 0,Y 312.564,Z 355.167,A -85,B 0,C 180,E1 -15463.004,E2 -15463.004} C_VEL
LIN {X 0,Y 312.671,Z 355.159,A -85,B 0,C 180,E1 -15465.685,E2 -15465.685} C_VEL
LIN {X 0,Y 312.671,Z 355.16,A -85,B 0,C 180,E1 -15469.641,E2 -15469.641} C_VEL
LIN {X 0,Y 312.78,Z 355.145,A -85,B 0,C 180,E1 -15472.252,E2 -15472.252} C_VEL
LIN {X 0,Y 312.675,Z 355.155,A -85,B 0,C 180,E1 -15474.842,E2 -15474.842} C_VEL
LIN {X 0,Y 312.952,Z 355.123,A -85,B 0,C 180,E1 -15478.713,E2 -15478.713} C_VEL
LIN {X 0,Y 312.967,Z 355.124,A -85,B 0,C 180,E1 -15481.287,E2 -15481.287} C_VEL
LIN {X 0,Y 312.827,Z 355.145,A -85,B 0,C 180,E1 -15486.45,E2 -15486.45} C_VEL
LIN {X 0,Y 312.736,Z 355.15,A -85,B 0,C 180,E1 -15489.051,E2 -15489.051} C_VEL
LIN {X 0,Y 312.617,Z 355.163,A -85,B 0,C 180,E1 -15492.992,E2 -15492.992} C_VEL
LIN {X 0,Y 312.612,Z 355.167,A -85,B 0,C 180,E1 -15495.651,E2 -15495.651} C_VEL
LIN {X 0,Y 312.524,Z 355.178,A -85,B 0,C 180,E1 -15499.713,E2 -15499.713} C_VEL
LIN {X 0,Y 312.5,Z 355.161,A -85,B 0,C 180,E1 -15502.776,E2 -15502.776} C_VEL
LIN {X 0,Y 312.47,Z 355.184,A -85,B 0,C 180,E1 -15506.733,E2 -15506.733} C_VEL
LIN {X 0,Y 312.455,Z 355.173,A -85,B 0,C 180,E1 -15509.659,E2 -15509.659} C_VEL
LIN {X 0,Y 312.508,Z 355.178,A -85,B 0,C 180,E1 -15513.69,E2 -15513.69} C_VEL
LIN {X 0,Y 312.498,Z 355.184,A -85,B 0,C 180,E1 -15517.389,E2 -15517.389} C_VEL
LIN {X 0,Y 312.429,Z 355.191,A -85,B 0,C 180,E1 -15520.719,E2 -15520.719} C_VEL
LIN {X 0,Y 312.439,Z 355.193,A -85,B 0,C 180,E1 -15524.212,E2 -15524.212} C_VEL
LIN {X 0,Y 312.444,Z 355.195,A -85,B 0,C 180,E1 -15527.927,E2 -15527.927} C_VEL
LIN {X 0,Y 312.467,Z 355.192,A -85,B 0,C 180,E1 -15531.926,E2 -15531.926} C_VEL
LIN {X 0,Y 312.525,Z 355.311,A -85,B 0,C 180,E1 -15533.88,E2 -15533.88} C_VEL
LIN {X 0,Y 315.221,Z 365.84,A -85,B 0,C 180,E1 -15537.274,E2 -15537.274} C_VEL
LIN {X 0,Y 316.138,Z 369.709,A -85,B 0,C 180,E1 -15538.447,E2 -15538.447} C_VEL
LIN {X 0,Y 325.536,Z 390.809,A -85,B 0,C 180,E1 -15539.984,E2 -15539.984} C_VEL
LIN {X 0,Y 327.751,Z 396.863,A -85,B 0,C 180,E1 -15540.356,E2 -15540.356} C_VEL
LIN {X 0,Y 330.618,Z 412.762,A -85,B 0,C 180,E1 -15541.025,E2 -15541.025} C_VEL
LIN {X 0,Y 327.974,Z 505.381,A -85,B 0,C 180,E1 -15543.044,E2 -15543.044} C_VEL
LIN {X 0,Y 327.002,Z 520.071,A -85,B 0,C 180,E1 -15543.56,E2 -15543.56} C_VEL
LIN {X 0,Y 325.607,Z 534.527,A -85,B 0,C 180,E1 -15544.342,E2 -15544.342} C_VEL
LIN {X 0,Y 324.053,Z 547.803,A -85,B 0,C 180,E1 -15545.326,E2 -15545.326} C_VEL
LIN {X 0,Y 322.336,Z 560.652,A -85,B 0,C 180,E1 -15546.562,E2 -15546.562} C_VEL
LIN {X 0,Y 320.472,Z 572.214,A -85,B 0,C 180,E1 -15547.944,E2 -15547.944} C_VEL
LIN {X 0,Y 318.669,Z 581.888,A -85,B 0,C 180,E1 -15549.339,E2 -15549.339} C_VEL
LIN {X 0,Y 316.728,Z 592.613,A -85,B 0,C 180,E1 -15551.234,E2 -15551.234} C_VEL
LIN {X 0,Y 315.048,Z 601.467,A -85,B 0,C 180,E1 -15553.144,E2 -15553.144} C_VEL
LIN {X 0,Y 313.579,Z 609.955,A -85,B 0,C 180,E1 -15555.398,E2 -15555.398} C_VEL
LIN {X 0,Y 312.351,Z 616.79,A -85,B 0,C 180,E1 -15557.66,E2 -15557.66} C_VEL
LIN {X 0,Y 311.602,Z 621.501,A -85,B 0,C 180,E1 -15559.607,E2 -15559.607} C_VEL
LIN {X 0,Y 311.013,Z 626.389,A -85,B 0,C 180,E1 -15562.21,E2 -15562.21} C_VEL
LIN {X 0,Y 310.718,Z 629.785,A -85,B 0,C 180,E1 -15564.811,E2 -15564.811} C_VEL
LIN {X 0,Y 310.649,Z 631.788,A -85,B 0,C 180,E1 -15567.409,E2 -15567.409} C_VEL
LIN {X 0,Y 310.616,Z 632.447,A -85,B 0,C 180,E1 -15570.002,E2 -15570.002} C_VEL
LIN {X 0,Y 310.65,Z 631.773,A -85,B 0,C 180,E1 -15572.595,E2 -15572.595} C_VEL
LIN {X 0,Y 310.723,Z 629.755,A -85,B 0,C 180,E1 -15575.193,E2 -15575.193} C_VEL
LIN {X 0,Y 311.028,Z 626.348,A -85,B 0,C 180,E1 -15577.794,E2 -15577.794} C_VEL
LIN {X 0,Y 311.606,Z 621.452,A -85,B 0,C 180,E1 -15580.397,E2 -15580.397} C_VEL
LIN {X 0,Y 312.354,Z 616.726,A -85,B 0,C 180,E1 -15582.344,E2 -15582.344} C_VEL
LIN {X 0,Y 313.577,Z 609.872,A -85,B 0,C 180,E1 -15584.606,E2 -15584.606} C_VEL
LIN {X 0,Y 315.044,Z 601.367,A -85,B 0,C 180,E1 -15586.86,E2 -15586.86} C_VEL
LIN {X 0,Y 316.718,Z 592.492,A -85,B 0,C 180,E1 -15588.771,E2 -15588.771} C_VEL
LIN {X 0,Y 318.666,Z 581.742,A -85,B 0,C 180,E1 -15590.665,E2 -15590.665} C_VEL
LIN {X 0,Y 320.659,Z 570.861,A -85,B 0,C 180,E1 -15592.216,E2 -15592.216} C_VEL
LIN {X 0,Y 322.663,Z 558.295,A -85,B 0,C 180,E1 -15593.672,E2 -15593.672} C_VEL
LIN {X 0,Y 324.277,Z 545.75,A -85,B 0,C 180,E1 -15594.831,E2 -15594.831} C_VEL
LIN {X 0,Y 325.864,Z 531.739,A -85,B 0,C 180,E1 -15595.812,E2 -15595.812} C_VEL
LIN {X 0,Y 327.159,Z 517.7,A -85,B 0,C 180,E1 -15596.516,E2 -15596.516} C_VEL
LIN {X 0,Y 328.021,Z 502.939,A -85,B 0,C 180,E1 -15596.999,E2 -15596.999} C_VEL
LIN {X 0,Y 329.441,Z 459.85,A -85,B 0,C 180,E1 -15597.949,E2 -15597.949} C_VEL
LIN {X 0,Y 334.344,Z 413.586,A -85,B 0,C 180,E1 -15599.782,E2 -15599.782} C_VEL
LIN {X 0,Y 333.756,Z 400.759,A -85,B 0,C 180,E1 -15600.762,E2 -15600.762} C_VEL
LIN {X 0,Y 332.74,Z 397.825,A -85,B 0,C 180,E1 -15601.225,E2 -15601.225} C_VEL
LIN {X 0,Y 331.671,Z 392.58,A -85,B 0,C 180,E1 -15602.291,E2 -15602.291} C_VEL
LIN {X 0,Y 329.784,Z 384.245,A -85,B 0,C 180,E1 -15604.387,E2 -15604.387} C_VEL
LIN {X 0,Y 327.385,Z 379.925,A -85,B 0,C 180,E1 -15606.346,E2 -15606.346} C_VEL
LIN {X 0,Y 325.001,Z 376.1,A -85,B 0,C 180,E1 -15608.878,E2 -15608.878} C_VEL
LIN {X 0,Y 323.846,Z 374.39,A -85,B 0,C 180,E1 -15610.623,E2 -15610.623} C_VEL
LIN {X 0,Y 322.955,Z 373.489,A -85,B 0,C 180,E1 -15612.426,E2 -15612.426} C_VEL
LIN {X 0,Y 322.515,Z 373.135,A -85,B 0,C 180,E1 -15614.214,E2 -15614.214} C_VEL
LIN {X 0,Y 322.491,Z 373.257,A -85,B 0,C 180,E1 -15615.988,E2 -15615.988} C_VEL
LIN {X 0,Y 322.83,Z 373.911,A -85,B 0,C 180,E1 -15617.749,E2 -15617.749} C_VEL
LIN {X 0,Y 323.76,Z 377.005,A -85,B 0,C 180,E1 -15620.986,E2 -15620.986} C_VEL
LIN {X 0,Y 324.783,Z 380.142,A -85,B 0,C 180,E1 -15623.194,E2 -15623.194} C_VEL
LIN {X 0,Y 326.323,Z 385.268,A -85,B 0,C 180,E1 -15625.947,E2 -15625.947} C_VEL
LIN {X 0,Y 327.25,Z 388.608,A -85,B 0,C 180,E1 -15627.346,E2 -15627.346} C_VEL
LIN {X 0,Y 330.475,Z 394.232,A -85,B 0,C 180,E1 -15628.736,E2 -15628.736} C_VEL
LIN {X 0,Y 334.325,Z 401.625,A -85,B 0,C 180,E1 -15630.225,E2 -15630.225} C_VEL
LIN {X 0,Y 336.974,Z 407.827,A -85,B 0,C 180,E1 -15631.21,E2 -15631.21} C_VEL
LIN {X 0,Y 338.662,Z 417.628,A -85,B 0,C 180,E1 -15632.139,E2 -15632.139} C_VEL
LIN {X 0,Y 330.89,Z 498.817,A -85,B 0,C 180,E1 -15635.198,E2 -15635.198} C_VEL
LIN {X 0,Y 329.353,Z 512.686,A -85,B 0,C 180,E1 -15635.998,E2 -15635.998} C_VEL
LIN {X 0,Y 327.592,Z 525.039,A -85,B 0,C 180,E1 -15636.951,E2 -15636.951} C_VEL
LIN {X 0,Y 325.682,Z 536.75,A -85,B 0,C 180,E1 -15638.115,E2 -15638.115} C_VEL
LIN {X 0,Y 323.628,Z 547.194,A -85,B 0,C 180,E1 -15639.392,E2 -15639.392} C_VEL
LIN {X 0,Y 321.587,Z 556.862,A -85,B 0,C 180,E1 -15640.864,E2 -15640.864} C_VEL
LIN {X 0,Y 319.246,Z 566.721,A -85,B 0,C 180,E1 -15642.711,E2 -15642.711} C_VEL
LIN {X 0,Y 317.316,Z 574.578,A -85,B 0,C 180,E1 -15644.587,E2 -15644.587} C_VEL
LIN {X 0,Y 315.643,Z 580.96,A -85,B 0,C 180,E1 -15646.48,E2 -15646.48} C_VEL
LIN {X 0,Y 314.208,Z 586.036,A -85,B 0,C 180,E1 -15648.387,E2 -15648.387} C_VEL
LIN {X 0,Y 313.165,Z 589.907,A -85,B 0,C 180,E1 -15650.31,E2 -15650.31} C_VEL
LIN {X 0,Y 312.3,Z 592.718,A -85,B 0,C 180,E1 -15652.24,E2 -15652.24} C_VEL
LIN {X 0,Y 311.754,Z 594.018,A -85,B 0,C 180,E1 -15653.528,E2 -15653.528} C_VEL
LIN {X 0,Y 311.437,Z 594.885,A -85,B 0,C 180,E1 -15654.821,E2 -15654.821} C_VEL
LIN {X 0,Y 311.268,Z 595.343,A -85,B 0,C 180,E1 -15656.116,E2 -15656.116} C_VEL
LIN {X 0,Y 311.077,Z 595.339,A -85,B 0,C 180,E1 -15657.41,E2 -15657.41} C_VEL
LIN {X 0,Y 310.913,Z 594.903,A -85,B 0,C 180,E1 -15658.705,E2 -15658.705} C_VEL
LIN {X 0,Y 310.81,Z 594.055,A -85,B 0,C 180,E1 -15660,E2 -15660} C_VEL
LIN {X 0,Y 310.787,Z 592.742,A -85,B 0,C 180,E1 -15661.296,E2 -15661.296} C_VEL
LIN {X 0,Y 310.889,Z 589.917,A -85,B 0,C 180,E1 -15663.24,E2 -15663.24} C_VEL
LIN {X 0,Y 311.008,Z 585.992,A -85,B 0,C 180,E1 -15665.186,E2 -15665.186} C_VEL
LIN {X 0,Y 311.334,Z 579.894,A -85,B 0,C 180,E1 -15667.458,E2 -15667.458} C_VEL
LIN {X 0,Y 311.726,Z 573.124,A -85,B 0,C 180,E1 -15669.408,E2 -15669.408} C_VEL
LIN {X 0,Y 312.345,Z 564.686,A -85,B 0,C 180,E1 -15671.355,E2 -15671.355} C_VEL
LIN {X 0,Y 313.014,Z 556.087,A -85,B 0,C 180,E1 -15672.975,E2 -15672.975} C_VEL
LIN {X 0,Y 313.804,Z 545.535,A -85,B 0,C 180,E1 -15674.593,E2 -15674.593} C_VEL
LIN {X 0,Y 314.512,Z 534.92,A -85,B 0,C 180,E1 -15675.924,E2 -15675.924} C_VEL
LIN {X 0,Y 315.314,Z 524.19,A -85,B 0,C 180,E1 -15677.01,E2 -15677.01} C_VEL
LIN {X 0,Y 316.07,Z 511.007,A -85,B 0,C 180,E1 -15678.054,E2 -15678.054} C_VEL
LIN {X 0,Y 316.705,Z 498.063,A -85,B 0,C 180,E1 -15678.812,E2 -15678.812} C_VEL
LIN {X 0,Y 317.281,Z 482.786,A -85,B 0,C 180,E1 -15679.406,E2 -15679.406} C_VEL
LIN {X 0,Y 319.603,Z 407.033,A -85,B 0,C 180,E1 -15681.825,E2 -15681.825} C_VEL
LIN {X 0,Y 316.095,Z 380.853,A -85,B 0,C 180,E1 -15682.865,E2 -15682.865} C_VEL
LIN {X 0,Y 316.274,Z 373.823,A -85,B 0,C 180,E1 -15684.343,E2 -15684.343} C_VEL
LIN {X 0,Y 313.398,Z 358.893,A -85,B 0,C 180,E1 -15687.695,E2 -15687.695} C_VEL
LIN {X 0,Y 312.623,Z 355.17,A -85,B 0,C 180,E1 -15688.587,E2 -15688.587} C_VEL
LIN {X 0,Y 312.511,Z 355.182,A -85,B 0,C 180,E1 -15692.666,E2 -15692.666} C_VEL
LIN {X 0,Y 312.541,Z 355.178,A -85,B 0,C 180,E1 -15695.949,E2 -15695.949} C_VEL
LIN {X 0,Y 312.461,Z 355.189,A -85,B 0,C 180,E1 -15700.114,E2 -15700.114} C_VEL
LIN {X 0,Y 312.464,Z 355.192,A -85,B 0,C 180,E1 -15703.964,E2 -15703.964} C_VEL
LIN {X 0,Y 312.461,Z 355.191,A -85,B 0,C 180,E1 -15707.924,E2 -15707.924} C_VEL
LIN {X 0,Y 312.489,Z 355.185,A -85,B 0,C 180,E1 -15711.922,E2 -15711.922} C_VEL
LIN {X 0,Y 312.553,Z 355.37,A -85,B 0,C 180,E1 -15715.306,E2 -15715.306} C_VEL
LIN {X 0,Y 314.887,Z 364.771,A -85,B 0,C 180,E1 -15718.385,E2 -15718.385} C_VEL
LIN {X 0,Y 323.526,Z 383.278,A -85,B 0,C 180,E1 -15719.793,E2 -15719.793} C_VEL
LIN {X 0,Y 329.491,Z 397.854,A -85,B 0,C 180,E1 -15720.754,E2 -15720.754} C_VEL
LIN {X 0,Y 330.807,Z 405.828,A -85,B 0,C 180,E1 -15721.077,E2 -15721.077} C_VEL
LIN {X 0,Y 327.951,Z 501.712,A -85,B 0,C 180,E1 -15723.167,E2 -15723.167} C_VEL
LIN {X 0,Y 327.086,Z 515.575,A -85,B 0,C 180,E1 -15723.692,E2 -15723.692} C_VEL
LIN {X 0,Y 325.86,Z 528.031,A -85,B 0,C 180,E1 -15724.359,E2 -15724.359} C_VEL
LIN {X 0,Y 324.391,Z 541.484,A -85,B 0,C 180,E1 -15725.349,E2 -15725.349} C_VEL
LIN {X 0,Y 322.766,Z 554.029,A -85,B 0,C 180,E1 -15726.541,E2 -15726.541} C_VEL
LIN {X 0,Y 320.846,Z 566.092,A -85,B 0,C 180,E1 -15727.967,E2 -15727.967} C_VEL
LIN {X 0,Y 318.713,Z 577.775,A -85,B 0,C 180,E1 -15729.676,E2 -15729.676} C_VEL
LIN {X 0,Y 316.753,Z 588.212,A -85,B 0,C 180,E1 -15731.567,E2 -15731.567} C_VEL
LIN {X 0,Y 315.121,Z 597.067,A -85,B 0,C 180,E1 -15733.539,E2 -15733.539} C_VEL
LIN {X 0,Y 313.756,Z 605.066,A -85,B 0,C 180,E1 -15735.734,E2 -15735.734} C_VEL
LIN {X 0,Y 312.594,Z 610.818,A -85,B 0,C 180,E1 -15737.666,E2 -15737.666} C_VEL
LIN {X 0,Y 311.878,Z 615.544,A -85,B 0,C 180,E1 -15739.612,E2 -15739.612} C_VEL
LIN {X 0,Y 311.192,Z 620.434,A -85,B 0,C 180,E1 -15742.21,E2 -15742.21} C_VEL
LIN {X 0,Y 310.836,Z 623.84,A -85,B 0,C 180,E1 -15744.809,E2 -15744.809} C_VEL
LIN {X 0,Y 310.687,Z 625.865,A -85,B 0,C 180,E1 -15747.405,E2 -15747.405} C_VEL
LIN {X 0,Y 310.618,Z 626.56,A -85,B 0,C 180,E1 -15749.998,E2 -15749.998} C_VEL
LIN {X 0,Y 310.685,Z 625.932,A -85,B 0,C 180,E1 -15752.591,E2 -15752.591} C_VEL
LIN {X 0,Y 310.823,Z 623.97,A -85,B 0,C 180,E1 -15755.187,E2 -15755.187} C_VEL
LIN {X 0,Y 311.165,Z 620.622,A -85,B 0,C 180,E1 -15757.786,E2 -15757.786} C_VEL
LIN {X 0,Y 311.853,Z 615.789,A -85,B 0,C 180,E1 -15760.385,E2 -15760.385} C_VEL
LIN {X 0,Y 312.895,Z 609.325,A -85,B 0,C 180,E1 -15762.978,E2 -15762.978} C_VEL
LIN {X 0,Y 314.266,Z 602.127,A -85,B 0,C 180,E1 -15765.232,E2 -15765.232} C_VEL
LIN {X 0,Y 315.608,Z 594.582,A -85,B 0,C 180,E1 -15767.158,E2 -15767.158} C_VEL
LIN {X 0,Y 317.333,Z 585.522,A -85,B 0,C 180,E1 -15769.065,E2 -15769.065} C_VEL
LIN {X 0,Y 319.367,Z 574.544,A -85,B 0,C 180,E1 -15770.95,E2 -15770.95} C_VEL
LIN {X 0,Y 321.345,Z 563.349,A -85,B 0,C 180,E1 -15772.501,E2 -15772.501} C_VEL
LIN {X 0,Y 323.216,Z 550.601,A -85,B 0,C 180,E1 -15773.927,E2 -15773.927} C_VEL
LIN {X 0,Y 324.954,Z 537.039,A -85,B 0,C 180,E1 -15775.113,E2 -15775.113} C_VEL
LIN {X 0,Y 326.441,Z 523.351,A -85,B 0,C 180,E1 -15776.016,E2 -15776.016} C_VEL
LIN {X 0,Y 327.53,Z 509.098,A -85,B 0,C 180,E1 -15776.694,E2 -15776.694} C_VEL
LIN {X 0,Y 328.266,Z 495.4,A -85,B 0,C 180,E1 -15777.102,E2 -15777.102} C_VEL
LIN {X 0,Y 328.709,Z 480.555,A -85,B 0,C 180,E1 -15777.423,E2 -15777.423} C_VEL
LIN {X 0,Y 328.318,Z 474.745,A -85,B 0,C 180,E1 -15777.599,E2 -15777.599} C_VEL
LIN {X 0,Y 323.808,Z 456.066,A -85,B 0,C 180,E1 -15778.478,E2 -15778.478} C_VEL
LIN {X 0,Y 323.345,Z 450.259,A -85,B 0,C 180,E1 -15778.667,E2 -15778.667} C_VEL
LIN {X 0,Y 324.537,Z 405.375,A -85,B 0,C 180,E1 -15779.666,E2 -15779.666} C_VEL
LIN {X 0,Y 323.271,Z 399.578,A -85,B 0,C 180,E1 -15779.939,E2 -15779.939} C_VEL
LIN {X 0,Y 315.864,Z 381.839,A -85,B 0,C 180,E1 -15781.179,E2 -15781.179} C_VEL
LIN {X 0,Y 309.096,Z 367.879,A -85,B 0,C 180,E1 -15782.317,E2 -15782.317} C_VEL
LIN {X 0,Y 307.667,Z 364.694,A -85,B 0,C 180,E1 -15782.599,E2 -15782.599} C_VEL
LIN {X 0,Y 305.474,Z 356.063,A -85,B 0,C 180,E1 -15785.614,E2 -15785.614} C_VEL
LIN {X 0,Y 305.409,Z 356.069,A -85,B 0,C 180,E1 -15788.519,E2 -15788.519} C_VEL
LIN {X 0,Y 305.425,Z 356.063,A -85,B 0,C 180,E1 -15792.579,E2 -15792.579} C_VEL
LIN {X 0,Y 305.412,Z 356.065,A -85,B 0,C 180,E1 -15796.342,E2 -15796.342} C_VEL
LIN {X 0,Y 305.4,Z 356.068,A -85,B 0,C 180,E1 -15799.883,E2 -15799.883} C_VEL
LIN {X 0,Y 305.452,Z 356.06,A -85,B 0,C 180,E1 -15803.635,E2 -15803.635} C_VEL
LIN {X 0,Y 305.453,Z 356.047,A -85,B 0,C 180,E1 -15806.482,E2 -15806.482} C_VEL
LIN {X 0,Y 305.417,Z 356.064,A -85,B 0,C 180,E1 -15809.586,E2 -15809.586} C_VEL
LIN {X 0,Y 305.441,Z 356.044,A -85,B 0,C 180,E1 -15812.601,E2 -15812.601} C_VEL
LIN {X 0,Y 305.46,Z 356.056,A -85,B 0,C 180,E1 -15815.535,E2 -15815.535} C_VEL
LIN {X 0,Y 305.47,Z 356.038,A -85,B 0,C 180,E1 -15819.811,E2 -15819.811} C_VEL
LIN {X 0,Y 305.537,Z 356.048,A -85,B 0,C 180,E1 -15823.977,E2 -15823.977} C_VEL
LIN {X 0,Y 305.571,Z 356.041,A -85,B 0,C 180,E1 -15826.703,E2 -15826.703} C_VEL
LIN {X 0,Y 305.739,Z 356.019,A -85,B 0,C 180,E1 -15831.261,E2 -15831.261} C_VEL
LIN {X 0,Y 305.769,Z 356.021,A -85,B 0,C 180,E1 -15833.401,E2 -15833.401} C_VEL
LIN {X 0,Y 305.844,Z 356.012,A -85,B 0,C 180,E1 -15837.366,E2 -15837.366} C_VEL
LIN {X 0,Y 305.898,Z 355.998,A -85,B 0,C 180,E1 -15840,E2 -15840} C_VEL
LIN {X 0,Y 305.841,Z 356.013,A -85,B 0,C 180,E1 -15842.634,E2 -15842.634} C_VEL
LIN {X 0,Y 305.772,Z 356.023,A -85,B 0,C 180,E1 -15846.599,E2 -15846.599} C_VEL
LIN {X 0,Y 305.68,Z 356.029,A -85,B 0,C 180,E1 -15849.261,E2 -15849.261} C_VEL
LIN {X 0,Y 305.571,Z 356.042,A -85,B 0,C 180,E1 -15853.297,E2 -15853.297} C_VEL
LIN {X 0,Y 305.54,Z 356.048,A -85,B 0,C 180,E1 -15856.023,E2 -15856.023} C_VEL
LIN {X 0,Y 305.47,Z 356.052,A -85,B 0,C 180,E1 -15860.188,E2 -15860.188} C_VEL
LIN {X 0,Y 305.426,Z 356.057,A -85,B 0,C 180,E1 -15864.468,E2 -15864.468} C_VEL
LIN {X 0,Y 305.428,Z 356.058,A -85,B 0,C 180,E1 -15867.4,E2 -15867.4} C_VEL
LIN {X 0,Y 305.404,Z 356.058,A -85,B 0,C 180,E1 -15870.415,E2 -15870.415} C_VEL
LIN {X 0,Y 305.452,Z 356.059,A -85,B 0,C 180,E1 -15874.079,E2 -15874.079} C_VEL
LIN {X 0,Y 305.44,Z 356.064,A -85,B 0,C 180,E1 -15876.744,E2 -15876.744} C_VEL
LIN {X 0,Y 305.398,Z 356.067,A -85,B 0,C 180,E1 -15880.591,E2 -15880.591} C_VEL
LIN {X 0,Y 305.41,Z 356.065,A -85,B 0,C 180,E1 -15883.658,E2 -15883.658} C_VEL
LIN {X 0,Y 305.424,Z 356.067,A -85,B 0,C 180,E1 -15887.421,E2 -15887.421} C_VEL
LIN {X 0,Y 305.432,Z 356.068,A -85,B 0,C 180,E1 -15891.594,E2 -15891.594} C_VEL
LIN {X 0,Y 305.502,Z 356.222,A -85,B 0,C 180,E1 -15893.216,E2 -15893.216} C_VEL
LIN {X 0,Y 308.294,Z 367.102,A -85,B 0,C 180,E1 -15896.834,E2 -15896.834} C_VEL
LIN {X 0,Y 308.825,Z 369.572,A -85,B 0,C 180,E1 -15897.608,E2 -15897.608} C_VEL
LIN {X 0,Y 318.659,Z 391.078,A -85,B 0,C 180,E1 -15899.275,E2 -15899.275} C_VEL
LIN {X 0,Y 321.823,Z 399.434,A -85,B 0,C 180,E1 -15899.82,E2 -15899.82} C_VEL
LIN {X 0,Y 324.407,Z 414.334,A -85,B 0,C 180,E1 -15900.456,E2 -15900.456} C_VEL
LIN {X 0,Y 321.614,Z 506.792,A -85,B 0,C 180,E1 -15902.51,E2 -15902.51} C_VEL
LIN {X 0,Y 320.603,Z 520.807,A -85,B 0,C 180,E1 -15903.034,E2 -15903.034} C_VEL
LIN {X 0,Y 319.238,Z 534.466,A -85,B 0,C 180,E1 -15903.792,E2 -15903.792} C_VEL
LIN {X 0,Y 317.601,Z 547.741,A -85,B 0,C 180,E1 -15904.79,E2 -15904.79} C_VEL
LIN {X 0,Y 315.961,Z 559.524,A -85,B 0,C 180,E1 -15905.93,E2 -15905.93} C_VEL
LIN {X 0,Y 313.896,Z 572.15,A -85,B 0,C 180,E1 -15907.457,E2 -15907.457} C_VEL
LIN {X 0,Y 311.999,Z 581.824,A -85,B 0,C 180,E1 -15908.877,E2 -15908.877} C_VEL
LIN {X 0,Y 309.966,Z 592.548,A -85,B 0,C 180,E1 -15910.808,E2 -15910.808} C_VEL
LIN {X 0,Y 308.207,Z 601.401,A -85,B 0,C 180,E1 -15912.759,E2 -15912.759} C_VEL
LIN {X 0,Y 306.642,Z 609.888,A -85,B 0,C 180,E1 -15915.06,E2 -15915.06} C_VEL
LIN {X 0,Y 305.378,Z 616.724,A -85,B 0,C 180,E1 -15917.373,E2 -15917.373} C_VEL
LIN {X 0,Y 304.592,Z 621.435,A -85,B 0,C 180,E1 -15919.365,E2 -15919.365} C_VEL
LIN {X 0,Y 303.95,Z 626.323,A -85,B 0,C 180,E1 -15922.028,E2 -15922.028} C_VEL
LIN {X 0,Y 303.636,Z 629.718,A -85,B 0,C 180,E1 -15924.69,E2 -15924.69} C_VEL
LIN {X 0,Y 303.575,Z 631.722,A -85,B 0,C 180,E1 -15927.348,E2 -15927.348} C_VEL
LIN {X 0,Y 303.532,Z 632.38,A -85,B 0,C 180,E1 -15930.002,E2 -15930.002} C_VEL
LIN {X 0,Y 303.576,Z 631.706,A -85,B 0,C 180,E1 -15932.656,E2 -15932.656} C_VEL
LIN {X 0,Y 303.638,Z 629.687,A -85,B 0,C 180,E1 -15935.314,E2 -15935.314} C_VEL
LIN {X 0,Y 303.982,Z 626.28,A -85,B 0,C 180,E1 -15937.976,E2 -15937.976} C_VEL
LIN {X 0,Y 304.595,Z 621.383,A -85,B 0,C 180,E1 -15940.639,E2 -15940.639} C_VEL
LIN {X 0,Y 305.382,Z 616.657,A -85,B 0,C 180,E1 -15942.631,E2 -15942.631} C_VEL
LIN {X 0,Y 306.639,Z 609.802,A -85,B 0,C 180,E1 -15944.944,E2 -15944.944} C_VEL
LIN {X 0,Y 308.209,Z 601.297,A -85,B 0,C 180,E1 -15947.245,E2 -15947.245} C_VEL
LIN {X 0,Y 309.957,Z 592.421,A -85,B 0,C 180,E1 -15949.196,E2 -15949.196} C_VEL
LIN {X 0,Y 311.998,Z 581.671,A -85,B 0,C 180,E1 -15951.127,E2 -15951.127} C_VEL
LIN {X 0,Y 314.081,Z 570.79,A -85,B 0,C 180,E1 -15952.707,E2 -15952.707} C_VEL
LIN {X 0,Y 316.049,Z 558.898,A -85,B 0,C 180,E1 -15954.116,E2 -15954.116} C_VEL
LIN {X 0,Y 317.827,Z 545.677,A -85,B 0,C 180,E1 -15955.37,E2 -15955.37} C_VEL
LIN {X 0,Y 319.505,Z 531.664,A -85,B 0,C 180,E1 -15956.365,E2 -15956.365} C_VEL
LIN {X 0,Y 320.83,Z 517.622,A -85,B 0,C 180,E1 -15957.081,E2 -15957.081} C_VEL
LIN {X 0,Y 321.717,Z 502.854,A -85,B 0,C 180,E1 -15957.573,E2 -15957.573} C_VEL
LIN {X 0,Y 322.561,Z 479.603,A -85,B 0,C 180,E1 -15958.112,E2 -15958.112} C_VEL
LIN {X 0,Y 329.911,Z 414.873,A -85,B 0,C 180,E1 -15960.724,E2 -15960.724} C_VEL
LIN {X 0,Y 329.582,Z 404.595,A -85,B 0,C 180,E1 -15961.528,E2 -15961.528} C_VEL
LIN {X 0,Y 327.071,Z 396.895,A -85,B 0,C 180,E1 -15962.875,E2 -15962.875} C_VEL
LIN {X 0,Y 325.41,Z 389.325,A -85,B 0,C 180,E1 -15964.845,E2 -15964.845} C_VEL
LIN {X 0,Y 323.439,Z 385.791,A -85,B 0,C 180,E1 -15966.489,E2 -15966.489} C_VEL
LIN {X 0,Y 320.685,Z 381.459,A -85,B 0,C 180,E1 -15969.463,E2 -15969.463} C_VEL
LIN {X 0,Y 319.357,Z 379.79,A -85,B 0,C 180,E1 -15971.563,E2 -15971.563} C_VEL
LIN {X 0,Y 318.654,Z 379.125,A -85,B 0,C 180,E1 -15973.296,E2 -15973.296} C_VEL
LIN {X 0,Y 318.315,Z 378.937,A -85,B 0,C 180,E1 -15975.048,E2 -15975.048} C_VEL
LIN {X 0,Y 318.375,Z 379.252,A -85,B 0,C 180,E1 -15976.818,E2 -15976.818} C_VEL
LIN {X 0,Y 318.595,Z 380.261,A -85,B 0,C 180,E1 -15978.594,E2 -15978.594} C_VEL
LIN {X 0,Y 319.052,Z 381.976,A -85,B 0,C 180,E1 -15980.443,E2 -15980.443} C_VEL
LIN {X 0,Y 319.905,Z 384.884,A -85,B 0,C 180,E1 -15982.726,E2 -15982.726} C_VEL
LIN {X 0,Y 321.214,Z 389.43,A -85,B 0,C 180,E1 -15985.305,E2 -15985.305} C_VEL
LIN {X 0,Y 324.682,Z 395.386,A -85,B 0,C 180,E1 -15987.119,E2 -15987.119} C_VEL
LIN {X 0,Y 327.399,Z 400.344,A -85,B 0,C 180,E1 -15988.352,E2 -15988.352} C_VEL
LIN {X 0,Y 330.828,Z 407.3,A -85,B 0,C 180,E1 -15989.77,E2 -15989.77} C_VEL
LIN {X 0,Y 332.717,Z 412.119,A -85,B 0,C 180,E1 -15990.545,E2 -15990.545} C_VEL
LIN {X 0,Y 333.873,Z 419.832,A -85,B 0,C 180,E1 -15991.295,E2 -15991.295} C_VEL
LIN {X 0,Y 325.601,Z 499.581,A -85,B 0,C 180,E1 -15994.382,E2 -15994.382} C_VEL
LIN {X 0,Y 323.906,Z 513.716,A -85,B 0,C 180,E1 -15995.226,E2 -15995.226} C_VEL
LIN {X 0,Y 322.034,Z 525.821,A -85,B 0,C 180,E1 -15996.188,E2 -15996.188} C_VEL
LIN {X 0,Y 319.688,Z 538.863,A -85,B 0,C 180,E1 -15997.528,E2 -15997.528} C_VEL
LIN {X 0,Y 317.317,Z 549.861,A -85,B 0,C 180,E1 -15998.963,E2 -15998.963} C_VEL
LIN {X 0,Y 315.163,Z 559.149,A -85,B 0,C 180,E1 -16000.458,E2 -16000.458} C_VEL
LIN {X 0,Y 312.697,Z 568.56,A -85,B 0,C 180,E1 -16002.337,E2 -16002.337} C_VEL
LIN {X 0,Y 310.659,Z 576.164,A -85,B 0,C 180,E1 -16004.248,E2 -16004.248} C_VEL
LIN {X 0,Y 308.887,Z 582.285,A -85,B 0,C 180,E1 -16006.178,E2 -16006.178} C_VEL
LIN {X 0,Y 307.34,Z 587.131,A -85,B 0,C 180,E1 -16008.123,E2 -16008.123} C_VEL
LIN {X 0,Y 306.239,Z 590.804,A -85,B 0,C 180,E1 -16010.089,E2 -16010.089} C_VEL
LIN {X 0,Y 305.314,Z 593.449,A -85,B 0,C 180,E1 -16012.061,E2 -16012.061} C_VEL
LIN {X 0,Y 304.744,Z 594.657,A -85,B 0,C 180,E1 -16013.379,E2 -16013.379} C_VEL
LIN {X 0,Y 304.391,Z 595.444,A -85,B 0,C 180,E1 -16014.701,E2 -16014.701} C_VEL
LIN {X 0,Y 304.193,Z 595.769,A -85,B 0,C 180,E1 -16016.026,E2 -16016.026} C_VEL
LIN {X 0,Y 303.993,Z 595.665,A -85,B 0,C 180,E1 -16017.35,E2 -16017.35} C_VEL
LIN {X 0,Y 303.823,Z 595.15,A -85,B 0,C 180,E1 -16018.675,E2 -16018.675} C_VEL
LIN {X 0,Y 303.719,Z 594.188,A -85,B 0,C 180,E1 -16020,E2 -16020} C_VEL
LIN {X 0,Y 303.699,Z 592.763,A -85,B 0,C 180,E1 -16021.326,E2 -16021.326} C_VEL
LIN {X 0,Y 303.818,Z 589.784,A -85,B 0,C 180,E1 -16023.315,E2 -16023.315} C_VEL
LIN {X 0,Y 303.92,Z 585.694,A -85,B 0,C 180,E1 -16025.307,E2 -16025.307} C_VEL
LIN {X 0,Y 304.22,Z 580.379,A -85,B 0,C 180,E1 -16027.3,E2 -16027.3} C_VEL
LIN {X 0,Y 304.589,Z 573.651,A -85,B 0,C 180,E1 -16029.295,E2 -16029.295} C_VEL
LIN {X 0,Y 305.213,Z 565.248,A -85,B 0,C 180,E1 -16031.287,E2 -16031.287} C_VEL
LIN {X 0,Y 305.859,Z 556.695,A -85,B 0,C 180,E1 -16032.946,E2 -16032.946} C_VEL
LIN {X 0,Y 306.664,Z 546.207,A -85,B 0,C 180,E1 -16034.602,E2 -16034.602} C_VEL
LIN {X 0,Y 307.429,Z 535.979,A -85,B 0,C 180,E1 -16035.922,E2 -16035.922} C_VEL
LIN {X 0,Y 308.24,Z 524.805,A -85,B 0,C 180,E1 -16037.095,E2 -16037.095} C_VEL
LIN {X 0,Y 309.034,Z 510.913,A -85,B 0,C 180,E1 -16038.222,E2 -16038.222} C_VEL
LIN {X 0,Y 309.678,Z 497.857,A -85,B 0,C 180,E1 -16038.998,E2 -16038.998} C_VEL
LIN {X 0,Y 310.278,Z 482.572,A -85,B 0,C 180,E1 -16039.604,E2 -16039.604} C_VEL
LIN {X 0,Y 312.601,Z 407.432,A -85,B 0,C 180,E1 -16042.086,E2 -16042.086} C_VEL
LIN {X 0,Y 309.174,Z 381.456,A -85,B 0,C 180,E1 -16043.131,E2 -16043.131} C_VEL
LIN {X 0,Y 309.334,Z 375.283,A -85,B 0,C 180,E1 -16044.399,E2 -16044.399} C_VEL
LIN {X 0,Y 306.577,Z 360.932,A -85,B 0,C 180,E1 -16047.659,E2 -16047.659} C_VEL
LIN {X 0,Y 305.568,Z 356.048,A -85,B 0,C 180,E1 -16048.787,E2 -16048.787} C_VEL
LIN {X 0,Y 305.472,Z 356.058,A -85,B 0,C 180,E1 -16053.516,E2 -16053.516} C_VEL
LIN {X 0,Y 305.459,Z 356.06,A -85,B 0,C 180,E1 -16056.742,E2 -16056.742} C_VEL
LIN {X 0,Y 305.415,Z 356.064,A -85,B 0,C 180,E1 -16060.589,E2 -16060.589} C_VEL
LIN {X 0,Y 305.428,Z 356.066,A -85,B 0,C 180,E1 -16063.655,E2 -16063.655} C_VEL
LIN {X 0,Y 305.442,Z 356.064,A -85,B 0,C 180,E1 -16067.417,E2 -16067.417} C_VEL
LIN {X 0,Y 305.465,Z 356.06,A -85,B 0,C 180,E1 -16071.594,E2 -16071.594} C_VEL
LIN {X 0,Y 305.498,Z 356.089,A -85,B 0,C 180,E1 -16074.587,E2 -16074.587} C_VEL
LIN {X 0,Y 307.738,Z 365.028,A -85,B 0,C 180,E1 -16077.566,E2 -16077.566} C_VEL
LIN {X 0,Y 316.564,Z 383.495,A -85,B 0,C 180,E1 -16079.059,E2 -16079.059} C_VEL
LIN {X 0,Y 323.485,Z 400.208,A -85,B 0,C 180,E1 -16080.214,E2 -16080.214} C_VEL
LIN {X 0,Y 324.557,Z 405.771,A -85,B 0,C 180,E1 -16080.461,E2 -16080.461} C_VEL
LIN {X 0,Y 321.838,Z 497.417,A -85,B 0,C 180,E1 -16082.483,E2 -16082.483} C_VEL
LIN {X 0,Y 321.077,Z 510.356,A -85,B 0,C 180,E1 -16082.897,E2 -16082.897} C_VEL
LIN {X 0,Y 319.999,Z 522.972,A -85,B 0,C 180,E1 -16083.504,E2 -16083.504} C_VEL
LIN {X 0,Y 318.651,Z 535.767,A -85,B 0,C 180,E1 -16084.35,E2 -16084.35} C_VEL
LIN {X 0,Y 317.035,Z 548.197,A -85,B 0,C 180,E1 -16085.418,E2 -16085.418} C_VEL
LIN {X 0,Y 315.302,Z 559.96,A -85,B 0,C 180,E1 -16086.692,E2 -16086.692} C_VEL
LIN {X 0,Y 313.215,Z 571.77,A -85,B 0,C 180,E1 -16088.268,E2 -16088.268} C_VEL
LIN {X 0,Y 311.339,Z 581.545,A -85,B 0,C 180,E1 -16089.862,E2 -16089.862} C_VEL
LIN {X 0,Y 309.403,Z 591.305,A -85,B 0,C 180,E1 -16091.799,E2 -16091.799} C_VEL
LIN {X 0,Y 307.979,Z 598.834,A -85,B 0,C 180,E1 -16093.609,E2 -16093.609} C_VEL
LIN {X 0,Y 306.627,Z 606.143,A -85,B 0,C 180,E1 -16095.734,E2 -16095.734} C_VEL
LIN {X 0,Y 305.336,Z 612.565,A -85,B 0,C 180,E1 -16098.042,E2 -16098.042} C_VEL
LIN {X 0,Y 304.431,Z 618.252,A -85,B 0,C 180,E1 -16100.698,E2 -16100.698} C_VEL
LIN {X 0,Y 303.922,Z 622.383,A -85,B 0,C 180,E1 -16103.359,E2 -16103.359} C_VEL
LIN {X 0,Y 303.673,Z 625.088,A -85,B 0,C 180,E1 -16106.017,E2 -16106.017} C_VEL
LIN {X 0,Y 303.538,Z 626.445,A -85,B 0,C 180,E1 -16108.671,E2 -16108.671} C_VEL
LIN {X 0,Y 303.537,Z 626.478,A -85,B 0,C 180,E1 -16111.325,E2 -16111.325} C_VEL
LIN {X 0,Y 303.668,Z 625.187,A -85,B 0,C 180,E1 -16113.979,E2 -16113.979} C_VEL
LIN {X 0,Y 303.914,Z 622.541,A -85,B 0,C 180,E1 -16116.638,E2 -16116.638} C_VEL
LIN {X 0,Y 304.419,Z 618.466,A -85,B 0,C 180,E1 -16119.298,E2 -16119.298} C_VEL
LIN {X 0,Y 305.306,Z 612.839,A -85,B 0,C 180,E1 -16121.955,E2 -16121.955} C_VEL
LIN {X 0,Y 306.586,Z 606.488,A -85,B 0,C 180,E1 -16124.264,E2 -16124.264} C_VEL
LIN {X 0,Y 307.946,Z 598.65,A -85,B 0,C 180,E1 -16126.557,E2 -16126.557} C_VEL
LIN {X 0,Y 309.648,Z 590.327,A -85,B 0,C 180,E1 -16128.525,E2 -16128.525} C_VEL
LIN {X 0,Y 311.622,Z 580.371,A -85,B 0,C 180,E1 -16130.459,E2 -16130.459} C_VEL
LIN {X 0,Y 313.727,Z 569.284,A -85,B 0,C 180,E1 -16132.209,E2 -16132.209} C_VEL
LIN {X 0,Y 315.679,Z 558.25,A -85,B 0,C 180,E1 -16133.622,E2 -16133.622} C_VEL
LIN {X 0,Y 317.399,Z 546.268,A -85,B 0,C 180,E1 -16134.877,E2 -16134.877} C_VEL
LIN {X 0,Y 319.037,Z 533.003,A -85,B 0,C 180,E1 -16135.963,E2 -16135.963} C_VEL
LIN {X 0,Y 320.454,Z 519.215,A -85,B 0,C 180,E1 -16136.803,E2 -16136.803} C_VEL
LIN {X 0,Y 321.509,Z 504.86,A -85,B 0,C 180,E1 -16137.411,E2 -16137.411} C_VEL
LIN {X 0,Y 322.279,Z 484.815,A -85,B 0,C 180,E1 -16137.913,E2 -16137.913} C_VEL
LIN {X 0,Y 323.345,Z 450.259,A -85,B 0,C 180,E1 -16138.667,E2 -16138.667} C_VEL
LIN {X 0,Y 322.875,Z 444.459,A -85,B 0,C 180,E1 -16138.857,E2 -16138.857} C_VEL
LIN {X 0,Y 318.404,Z 425.827,A -85,B 0,C 180,E1 -16139.775,E2 -16139.775} C_VEL
LIN {X 0,Y 318.051,Z 420.026,A -85,B 0,C 180,E1 -16139.96,E2 -16139.96} C_VEL
LIN {X 0,Y 318.378,Z 406.562,A -85,B 0,C 180,E1 -16140.27,E2 -16140.27} C_VEL
LIN {X 0,Y 317.223,Z 401.835,A -85,B 0,C 180,E1 -16140.514,E2 -16140.514} C_VEL
LIN {X 0,Y 310.07,Z 384.658,A -85,B 0,C 180,E1 -16141.754,E2 -16141.754} C_VEL
LIN {X 0,Y 302.014,Z 368.156,A -85,B 0,C 180,E1 -16143.165,E2 -16143.165} C_VEL
LIN {X 0,Y 300.429,Z 364.805,A -85,B 0,C 180,E1 -16143.475,E2 -16143.475} C_VEL
LIN {X 0,Y 298.429,Z 356.938,A -85,B 0,C 180,E1 -16146.296,E2 -16146.296} C_VEL
LIN {X 0,Y 298.341,Z 356.947,A -85,B 0,C 180,E1 -16149.494,E2 -16149.494} C_VEL
LIN {X 0,Y 298.361,Z 356.944,A -85,B 0,C 180,E1 -16153.095,E2 -16153.095} C_VEL
LIN {X 0,Y 298.361,Z 356.944,A -85,B 0,C 180,E1 -16156.913,E2 -16156.913} C_VEL
LIN {X 0,Y 298.374,Z 356.934,A -85,B 0,C 180,E1 -16161.009,E2 -16161.009} C_VEL
LIN {X 0,Y 298.394,Z 356.939,A -85,B 0,C 180,E1 -16163.927,E2 -16163.927} C_VEL
LIN {X 0,Y 298.381,Z 356.923,A -85,B 0,C 180,E1 -16167.198,E2 -16167.198} C_VEL
LIN {X 0,Y 298.389,Z 356.943,A -85,B 0,C 180,E1 -16170.624,E2 -16170.624} C_VEL
LIN {X 0,Y 298.425,Z 356.921,A -85,B 0,C 180,E1 -16174.918,E2 -16174.918} C_VEL
LIN {X 0,Y 298.388,Z 356.94,A -85,B 0,C 180,E1 -16177.861,E2 -16177.861} C_VEL
LIN {X 0,Y 298.451,Z 356.906,A -85,B 0,C 180,E1 -16180.751,E2 -16180.751} C_VEL
LIN {X 0,Y 298.573,Z 356.918,A -85,B 0,C 180,E1 -16184.994,E2 -16184.994} C_VEL
LIN {X 0,Y 298.569,Z 356.918,A -85,B 0,C 180,E1 -16189.146,E2 -16189.146} C_VEL
LIN {X 0,Y 298.682,Z 356.899,A -85,B 0,C 180,E1 -16191.884,E2 -16191.884} C_VEL
LIN {X 0,Y 298.614,Z 356.908,A -85,B 0,C 180,E1 -16194.598,E2 -16194.598} C_VEL
LIN {X 0,Y 298.889,Z 356.876,A -85,B 0,C 180,E1 -16198.653,E2 -16198.653} C_VEL
LIN {X 0,Y 298.9,Z 356.876,A -85,B 0,C 180,E1 -16201.347,E2 -16201.347} C_VEL
LIN {X 0,Y 298.72,Z 356.9,A -85,B 0,C 180,E1 -16206.756,E2 -16206.756} C_VEL
LIN {X 0,Y 298.611,Z 356.91,A -85,B 0,C 180,E1 -16209.483,E2 -16209.483} C_VEL
LIN {X 0,Y 298.53,Z 356.919,A -85,B 0,C 180,E1 -16213.616,E2 -16213.616} C_VEL
LIN {X 0,Y 298.473,Z 356.926,A -85,B 0,C 180,E1 -16216.413,E2 -16216.413} C_VEL
LIN {X 0,Y 298.428,Z 356.934,A -85,B 0,C 180,E1 -16219.618,E2 -16219.618} C_VEL
LIN {X 0,Y 298.368,Z 356.928,A -85,B 0,C 180,E1 -16223.605,E2 -16223.605} C_VEL
LIN {X 0,Y 298.388,Z 356.939,A -85,B 0,C 180,E1 -16226.584,E2 -16226.584} C_VEL
LIN {X 0,Y 298.344,Z 356.93,A -85,B 0,C 180,E1 -16229.649,E2 -16229.649} C_VEL
LIN {X 0,Y 298.38,Z 356.939,A -85,B 0,C 180,E1 -16232.802,E2 -16232.802} C_VEL
LIN {X 0,Y 298.414,Z 356.939,A -85,B 0,C 180,E1 -16236.804,E2 -16236.804} C_VEL
LIN {X 0,Y 298.362,Z 356.944,A -85,B 0,C 180,E1 -16239.494,E2 -16239.494} C_VEL
LIN {X 0,Y 298.359,Z 356.944,A -85,B 0,C 180,E1 -16243.099,E2 -16243.099} C_VEL
LIN {X 0,Y 298.36,Z 356.948,A -85,B 0,C 180,E1 -16246.916,E2 -16246.916} C_VEL
LIN {X 0,Y 298.376,Z 356.946,A -85,B 0,C 180,E1 -16251.013,E2 -16251.013} C_VEL
LIN {X 0,Y 298.445,Z 357.149,A -85,B 0,C 180,E1 -16252.514,E2 -16252.514} C_VEL
LIN {X 0,Y 301.039,Z 367.024,A -85,B 0,C 180,E1 -16255.926,E2 -16255.926} C_VEL
LIN {X 0,Y 301.669,Z 369.571,A -85,B 0,C 180,E1 -16256.743,E2 -16256.743} C_VEL
LIN {X 0,Y 311.206,Z 390.11,A -85,B 0,C 180,E1 -16258.432,E2 -16258.432} C_VEL
LIN {X 0,Y 315.866,Z 401.561,A -85,B 0,C 180,E1 -16259.246,E2 -16259.246} C_VEL
